(* der ausgabestring muss nochg mit 0 abgeschlossen werden *)
pt^ := 0;

(* revision history
hm		9.6.2007	rev 1.0		
	original version

hm		15.dec 2007	rev 1.1
	changed code for better performance

hm	29. mar. 2008	rev 1.2
	changed STRING to STRING(32)

hm	20. jun. 2008	rev 1.3
	performance improvement

*)

END_FUNCTION

// oscat_basic/POUs/String/DWORD_TO_STRF
FUNCTION DWORD_TO_STRF : STRING(20)
VAR_INPUT
	IN : DWORD;
	N : INT;
END_VAR


(*
version 1.0	26 jan 2007
programmer 	hugo
tested by		tobias

dword_to_strF converts a DWORD, BYTE or Word to a fixed length String.
the string will be filled with leading zeroes to achieve the fixed length, or if too long, the lowest digits will be used.
the maximum allowed length is 20 mdigits.

for example:	dword_to_strf(123,4) = '0123' 
				dword_to_strf(123,2) = '23'
*)

(* limit N to max 20 characters *)
(* convert dword to string first and cut to length N *)
DWORD_TO_STRF := FIX(DWORD_TO_STRING(in),LIMIT(0,N,20),48,1);


(* revision history
hm	26. jan.2007	rev 1.0		
	original version

hm	29. mar. 2008	rev 1.1
	changed STRING to STRING(20)
	limit the output string to max 20 digits
*)

END_FUNCTION

// oscat_basic/POUs/String/FIX
FUNCTION FIX : STRING(STRING_LENGTH)
VAR_INPUT
	str : STRING(STRING_LENGTH);
	L : INT;
	C : BYTE;
	M : INT;
END_VAR
VAR
	N : INT;
	SX: STRING(STRING_LENGTH);
END_VAR

(*
version 1.0	29. mar. 2008
programmer 	hugo
tested by	tobias

the function fix truncates a string at length L 
or if the string is shorter then L it will be filled with ending Spaces till its length = N.

*)

(* make sure L does not exceed the limits of a string *)
N := LIMIT(0,L,STRING_LENGTH) - LEN(str);
IF N <= 0 THEN
	(* truncate the string at length N *)
	IF M = 1 THEN
		FIX := RIGHT(str,L);
	ELSE
		FIX := LEFT(str,L);
	END_IF;
ELSIF M = 1 THEN
	(* connect fill characters at the beginning *)
	sx := FILL(C,N);
	FIX := CONCAT(sx,str);
ELSIF M = 2 THEN
	(* center str beween fill characters *)
	(* for an uneven number of fill characters, there is one more at the end *)
	sx := FILL(C,SHR(N+1,1));
	FIX := CONCAT(str,sx);
	SX := LEFT(sx,SHR(N,1));
	FIX := CONCAT(sx,FIX);
ELSE
	(* connect fill characters at the end *)
	SX := FILL(C,N);
	FIX := CONCAT(str,SX);
END_IF;


(* revision histroy
hm	29. mar. 2008	rev 1.0
	original release

*)

END_FUNCTION

// oscat_basic/POUs/String/DWORD_TO_STRH
FUNCTION DWORD_TO_STRH : STRING(8)
VAR_INPUT
	IN : DWORD;
END_VAR
VAR
	i : INT;
	temp : BYTE;
	pt : POINTER TO BYTE;
END_VAR

(*
version 1.3	29. mar. 2008
programmer 	hugo
tested by	tobias

DWORD_TO_STRINGH converts a DWORD to a String of Hexadecimal represented by '0' .. '9' and 'A' .. 'F'.
The lowest order Character will be on the right and the high order Character on the left.

*)

(* read output adress to pointer *)
pt := ADR(DWORD_TO_STRH) + 8;
(* wirte the closing byte for the string *)
pt^:= 0;

(* write the 8 hex characters backwards *)
FOR i := 1 TO 8 DO;
	(* decrement the pointer *)
	pt := pt - 1;
	(* read the lowest order hex value *)
	temp := DWORD_TO_BYTE(in AND 16#0000000F);
	(* convert value to hex character *)
	IF temp <= 9 THEN temp := temp + 48; ELSE temp := temp + 55; END_IF;
	(* write character to output string *)
	PT^ := temp;
	(* shift in for nect hex character *)
	in := SHR(in,4);
END_FOR;


(* code beofre rev 1.2
FOR i := 1 TO 8 DO
	X := DWORD_TO_BYTE(in AND 2#1111);
	IF X <= 9 THEN X := X + 48; ELSE X := X + 55; END_IF;
	Cx := CHR(X);
	temp := CONCAT(Cx, temp);
	in := SHR(in,4);
END_FOR;
DWORD_TO_STRH := temp;
*)


(* revision history
hm	9. jun. 2007	rev 1.0		
	original version 

hm	11. sep. 2007	rev 1.1
	changed coding for compatibility with twincat, concat cannot support a function as an argument.

hm	15. dec. 2007	rev 1.2
	changed code for better performance

hm	29. mar. 2008	rev 1.3
	changed STRING to STRING(8)

*)

END_FUNCTION

// oscat_basic/POUs/String/EXEC
FUNCTION EXEC : STRING(STRING_LENGTH)
VAR_INPUT
	str : STRING(STRING_LENGTH);
END_VAR
VAR
	pos: INT;
	R1: REAL;
	R2: REAL;
	operator: STRING(10);
END_VAR

(*
version 1.4	29. mar. 2008
programmer 	hugo
tested by		tobias

exec executes a mathematical term and returns the result as a string
the term can only be a simple term without brackets and only one operator
allowed operastors are: (+, -, *, /, ^, sqrt, sin, cos, tan).

*)

(* extract both numbers and operator *)
EXEC := UPPERCASE(TRIM(str));

pos := FINDB_NONUM(EXEC);
IF pos > 1 THEN R1 := STRING_TO_REAL(LEFT(EXEC,pos-1)); END_IF;
R2 := STRING_TO_REAL(RIGHT(EXEC,LEN(EXEC)-pos));
EXEC := LEFT(EXEC,pos);
pos := FINDB_NUM(EXEC);
operator := RIGHT(EXEC,LEN(EXEC) - pos);
IF operator = '' AND LEN(str) = 0 THEN
	EXEC := '';
	RETURN;
ELSIF operator = '' THEN
	EXEC := str;
	RETURN;
END_IF;
IF operator = '^' THEN
	EXEC := REAL_TO_STRING(EXPT(R1, R2));
ELSIF operator = 'SQRT' THEN
	EXEC := REAL_TO_STRING(SQRT(R2));
ELSIF operator = 'SIN' THEN
	EXEC := REAL_TO_STRING(SIN(r2));
ELSIF operator = 'COS' THEN
	EXEC := REAL_TO_STRING(COS(r2));
ELSIF operator = 'TAN' THEN
	EXEC := REAL_TO_STRING(TAN(R2));
ELSIF operator = '*' THEN
	EXEC := REAL_TO_STRING(R1 * R2);
ELSIF operator = '/' THEN
	IF R2 <> 0 THEN EXEC := REAL_TO_STRING(R1 / R2); ELSE EXEC := 'ERROR'; END_IF;
ELSIF operator = '+' THEN
	EXEC := REAL_TO_STRING(r1 + r2);
ELSIF operator = '-' THEN
	EXEC := REAL_TO_STRING(r1 - r2);
ELSE
	EXEC := 'ERROR';
END_IF;

IF EXEC = 'ERROR' THEN
	RETURN;
(* some systems deliver integer instead of real *)
ELSIF FIND(EXEC,'.') = 0 THEN
	EXEC := CONCAT(EXEC, '.0');
(* some systems deliver n. instead of n.0 ! *)
ELSIF RIGHT(EXEC,1) = '.' THEN
	EXEC := CONCAT(EXEC,'0');
END_IF;


(* revision history

hm 	6.feb 2007		rev 1.1
	cos has to be written in uppercase
	divide by 0 will return an error

hm	5. mar. 2008	rev 1.2
	add a 0 to the string if a '.' is at the end of the string

hm	20. mar. 2008	rev 1.3
	make sure the function always returns a real value in the form of x.y

hm	29. mar. 2008	rev 1.4
	changed STRING to STRING(STRING_LENGTH)
*)

END_FUNCTION

// oscat_basic/POUs/String/TRIM
FUNCTION TRIM : STRING(STRING_LENGTH)
VAR_INPUT
	str : STRING(STRING_LENGTH);
END_VAR
VAR
	pos: INT;
END_VAR

(*
version 1.2	29. mar. 2008
programmer 	hugo
tested by	tobias

the function deletes all blanks within a string.

*)

TRIM := str;
REPEAT
	pos := FIND(trim,' ');
	IF pos > 0 THEN TRIM := REPLACE(TRIM,'',1,pos); END_IF;
UNTIL pos = 0	END_REPEAT;


(* revision histroy
hm	6.10.2006		rev 1.0
	original release

hm	20. mar. 2008	rev 1.1
	avoid to call replace with pos = 0 because some systems will produce an error

hm	29. mar. 2008	rev 1.2
	changed STRING to STRING(STRING_LENGTH)
*)

END_FUNCTION

// oscat_basic/POUs/String/FINDB_NONUM
FUNCTION FINDB_NONUM : INT
VAR_INPUT
	str : STRING(STRING_LENGTH);
END_VAR
VAR
	pos: INT;
	pt : POINTER TO BYTE;
END_VAR

(*
version 1.3	21. oct. 2008
programmer 	hugo
tested by	oscat

findB_noNum searches str backwards and returns the last position which is not a number.
a number is characterized by a letter "0..9" or "."

*)

pt := ADR(str) + LEN(str) - 1;
FOR pos := LEN(str) TO 1 BY -1 DO;
	IF (PT^ < 48 AND PT^ <> 46) OR PT^ > 57 THEN
		FINDB_NONUM := pos;
		RETURN;
	END_IF;
	PT := PT - 1;
END_FOR;
FINDB_NONUM := 0;


(* revision history
hm	6. oct 2006		rev 1.0
	original version

hm	29. feb 2008	rev 1.1
	improved performance

hm	29. mar. 2008	rev 1.2
	changed STRING to STRING(STRING_LENGTH)

hm	21. oct. 2008	rev 1.3
	optimized code
*)

END_FUNCTION

// oscat_basic/POUs/String/FINDB_NUM
FUNCTION FINDB_NUM : INT
VAR_INPUT
	str : STRING(STRING_LENGTH);
END_VAR
VAR
	pos: INT;
	pt : POINTER TO BYTE;
END_VAR

(*
version 1.2	29. mar. 2008
programmer 	hugo
tested by	tobias

findB_Num searches str backward and returns the last position of a number
a number is characterized by a letter "0..9" or "."

*)

pt := ADR(str) + LEN(str) - 1;
FOR pos := LEN(str) TO 1 BY -1 DO;
	IF (PT^ > 47 AND PT^ < 58) OR PT^ = 46 THEN
		FINDB_NUM := pos;
		RETURN;
	END_IF;
	PT := PT - 1;
END_FOR;
FINDB_NUM := 0;

(* revision history
hm	6. oct 2006		rev 1.0
	original version

hm	29. feb 2008	rev 1.1
	improved performance

hm	29. mar. 2008	rev 1.2
	changed STRING to STRING(STRING_LENGTH)
*)

END_FUNCTION

// oscat_basic/POUs/String/FIND_CHAR
FUNCTION FIND_CHAR : INT
VAR_INPUT
	str : STRING(STRING_LENGTH);
	pos : INT;
END_VAR
VAR
	i: INT;
	pt : POINTER TO ARRAY[1..255] OF BYTE;
	stop: INT;
	X: BYTE;
END_VAR

(*
version 1.3	21. oct. 2008
programmer 	hugo
tested by	tobias

find_char searches str and returns the starting position of the first character that is not a control character.
control characters are the ascii character 00 .. 31 and 127

*)

pt := ADR(str);
stop := LEN(str);
FOR i := MAX(pos,1) TO stop DO;
	X := pt^[i];
	IF X > 31 AND ((setup.EXTENDED_ASCII AND X <> 127) OR (NOT setup.EXTENDED_ASCII AND X < 127)) THEN
		FIND_CHAR := i;
		RETURN;
	END_IF;
END_FOR;
FIND_CHAR := 0;


(* revision history
hm	29. feb 2008	rev 1.0
	original version

hm	26. mar. 2008	rev 1.1
	char will now accept extended ascii

hm	29. mar. 2008	rev 1.2
	changed STRING to STRING(STRING_LENGTH)

hm	21. oct. 2008	rev 1.3
	changes setup constants
	optimized code
*)

END_FUNCTION

// oscat_basic/POUs/String/FIND_CTRL
FUNCTION FIND_CTRL : INT
VAR_INPUT
	str : STRING(STRING_LENGTH);
	pos : INT;
END_VAR
VAR
	i: INT;
	pt : POINTER TO ARRAY[1..255] OF BYTE;
	stop: INT;
	x: BYTE;
END_VAR

(*
version 1.2	29. mar. 2008
programmer 	hugo
tested by		tobias

find_ctrl searches str and returns the starting position of a control character
control characters are the ascii character 00 .. 31 and 127.

*)

pt := ADR(str);
stop := LEN(str);
FOR i := MAX(pos,1) TO stop DO;
	x := PT^[I];
	IF x < 32 OR X = 127 THEN
		FIND_CTRL := i;
		RETURN;
	END_IF;
END_FOR;
FIND_CTRL := 0;


(* revision history
hm	29. feb 2008	rev 1.0
	original version

hm	26. mar. 2008	rev 1.1
	character 127 is now recognized as control

hm	29. mar. 2008	rev 1.2
	changed STRING to STRING(STRING_LENGTH)
*)

END_FUNCTION

// oscat_basic/POUs/String/FIND_NONUM
FUNCTION FIND_NONUM : INT
VAR_INPUT
	str : STRING(STRING_LENGTH);
	pos : INT;
END_VAR
VAR
	i: INT;
	pt : POINTER TO ARRAY[1..255] OF BYTE;
	end: INT;
	X: BYTE;
END_VAR

(*
version 1.3	21. oct. 2008
programmer 	hugo
tested by	tobias

find_noNum searches str and returns the first position which is not a number.
a number is characterized by a letter "0..9" or "."

*)

pt := ADR(str);
end := LEN(str);
FOR i := MAX(pos,1) TO end DO;
	X := pt^[i];
	IF (X < 48 AND X <> 46) OR X > 57 THEN
		FIND_NONUM := i;
		RETURN;
	END_IF;
END_FOR;
FIND_NONUM := 0;


(* revision history
hm	6. oct. 2006	rev 1.0
	original version

hm	29. feb 2008	rev 1.1
	added input pos to start search at position

hm	29. mar. 2008	rev 1.2
	changed STRING to STRING(STRING_LENGTH)

hm	21. oct. 2008	rev 1.3
	optimized code

*)

END_FUNCTION

// oscat_basic/POUs/String/FIND_NUM
FUNCTION FIND_NUM : INT
VAR_INPUT
	str : STRING(STRING_LENGTH);
	pos : INT;
END_VAR
VAR
	i : INT;
	pt : POINTER TO ARRAY[1..255] OF BYTE;
	stop : INT;
	X: BYTE;
END_VAR

(*
version 1.2	29. mar. 2008
programmer 	hugo
tested by		tobias

find_Num searches str and returns the starting position of a number
a number is characterized by a letter "0..9" or "."

*)

pt := ADR(str);
stop := LEN(str);
FOR i := MAX(pos,1) TO stop DO;
	X := pt^[i];
	IF (X > 47 AND X < 58) OR X = 46 THEN
		FIND_NUM := i;
		RETURN;
	END_IF;
END_FOR;
FIND_NUM := 0;


(* revision history
hm	6. oct. 2006	rev 1.0
	original version

hm	29. feb 2008	rev 1.1
	added input pos to start search at position

hm	29. mar. 2008	rev 1.2
	changed STRING to STRING(STRING_LENGTH)

*)

END_FUNCTION

// oscat_basic/POUs/String/FINDB
FUNCTION FINDB : INT
VAR_INPUT
	str1 : STRING(STRING_LENGTH);
	str2 : STRING(STRING_LENGTH);
END_VAR
VAR
	pos: INT;
	length: INT;
END_VAR

(*
version 1.3	29. mar. 2008
programmer 	hugo
tested by		tobias

the function find searches an str1 for the presence of str2 and returns the first position of str1 of the last presence in instring.
the function is similar to find except it searches from the right to left.
 a 0 is returned if the string is not found.

*)

length := LEN(str2);
FOR pos := LEN(str1) - length + 1 TO 1 BY -1 DO
	IF MID(str1,length,pos) = str2 THEN
		FindB := pos;
		RETURN;
	END_IF;
END_FOR;
FindB := 0;

(* revision history
hm	6. oct 2006		rev 1.0
	original version

hm	15 dec 2007		rev 1.1
	changed code for better performance

hm	29. feb 2008	rev 1.2
	added findb := 0 for compatibility reasons

hm	29. mar. 2008	rev 1.3
	changed STRING to STRING(STRING_LENGTH)
*)

END_FUNCTION

// oscat_basic/POUs/String/FINDP
FUNCTION FINDP : INT
VAR_INPUT
	str : STRING(STRING_LENGTH);
	src : STRING(STRING_LENGTH);
	pos: INT;
END_VAR
VAR
	i: INT;
	ls: INT;
	lx: INT;
	stp: INT;
END_VAR

(*
version 1.2	29. mar. 2008
programmer 	hugo
tested by	tobias

the function findP searches a string str for the occurence of src beginning at the position pos.

*)

ls := LEN(str);
lx := LEN(src);
IF ls < lx OR lx = 0 THEN RETURN; END_IF;
stp := ls - lx + 1;
FOR i := MAX(pos,1) TO stp DO
	IF MID(str,lx,i) = src THEN
		FINDP := i;
		RETURN;
	END_IF;
END_FOR;
FINDP := 0;

(* revision histroy
hm	4. feb. 2008	rev 1.0
	original release

hm	29. feb 2008	rev 1.1
	ADDED MAX(pos,1) in loop initialization

hm	29. mar. 2008	rev 1.2
	changed STRING to STRING(STRING_LENGTH)
*)

END_FUNCTION

// oscat_basic/POUs/String/FLOAT_TO_REAL
FUNCTION FLOAT_TO_REAL : REAL
VAR_INPUT
	FLT : STRING(20);
END_VAR
VAR
	pt : POINTER TO ARRAY[1..20] OF BYTE;
	i: INT;
	X: BYTE;
	sign: INT := 1;
	stop: INT;
	tmp: DINT;
	d : INT;
END_VAR

(*
version 1.3	23. oct. 2008
programmer 	hugo
tested by	oscat

FLOAT_TO_REAL converts a string to a REAL.
the function ignores all wrong characters.
the comma can be , or .
the exponent has to start with capital E or lowercase e .


*)

pt := ADR(FLT);
stop := LEN(FLT);

(* we first check for sign and exit if first number or dot is reached *)
FOR i := 1 TO stop DO
	X := pt^[i];
	IF X > 47 AND X < 58 OR X = 46 THEN
		EXIT;
	ELSIF X = 45 THEN
		(* code 45 is sign *)
		sign := -1;
	END_IF;
END_FOR;

(* now we scan numbers till end or dot or E is reached *)
FOR i := i TO stop DO
	X := pt^[i];
	IF X = 44 OR X = 46 OR X = 69 OR X = 101 THEN
		EXIT;
	(* calculate the value of the digit *)
	ELSIF X > 47 AND x < 58 THEN
		tmp := tmp * 10 + X - 48;
	END_IF;
END_FOR;

(* process the portion after the comma if comma or dot is reached exit if exponent starts *)
IF x = 44 OR X = 46 THEN
	FOR i := i + 1 TO stop DO
		X := pt^[i];
		IF X = 69 OR X = 101 THEN
			EXIT;
		ELSIF x > 47 AND x < 58 THEN
			tmp := tmp * 10 + X - 48;
			d := d - 1;
		END_IF;
	END_FOR;
END_IF;

(* process exponent if present *)
IF X = 69 OR X = 101 THEN
	d := d + DEC_TO_INT(RIGHT(FLT, stop - i));
END_IF;

FLOAT_TO_REAL :=  EXPN(10, d) * DINT_TO_REAL(TMP * SIGN);




(* revision histroy
hm	22. jun. 2008	rev 1.0
	original release

hm	2. oct. 2008	rev 1.1
	fixed an error, characters 8 and 9 would not be converted

hm	22. oct. 2008	rev 1.2
	last fix was not done correctly

hm	23. oct. 2008	rev 1.3
	optimzed code
*)

END_FUNCTION

// oscat_basic/POUs/String/FSTRING_TO_BYTE
FUNCTION FSTRING_TO_BYTE : BYTE
VAR_INPUT
	IN : STRING(12);
END_VAR


(*
version 1.1	20. sep. 2008
programmer 	hugo
tested by		oscat

FSTRING_TO_BYTE converts a formatted string into a byte.
the string can be of the form 2#01010, 8#7234, 16#2AD3 and 1234

*)

IF LEFT(IN, 2) = '2#' THEN
	(* we need to convert binary *)
	FSTRING_TO_BYTE := BIN_TO_BYTE(RIGHT(in, LEN(in) - 2));
ELSIF LEFT(in, 2) = '8#' THEN
	(* weneed to convert octals *)
	FSTRING_TO_BYTE := OCT_TO_BYTE(RIGHT(in, LEN(in) - 2));
ELSIF LEFT(in, 3) = '16#' THEN
	(* we need to convert hexadecimal *)
	FSTRING_TO_BYTE := HEX_TO_BYTE(RIGHT(in, LEN(in) - 3));
ELSE
	(* we assume decimal representation *)
	FSTRING_TO_BYTE := DEC_TO_BYTE(CLEAN(in,'0123456789'));
END_IF;


(* revision histroy
hm	18. jun. 2008	rev 1.0
	original release

hm	20. sep. 2008	rev 1.1
	changed length of input string from 20 to 12
*)

END_FUNCTION

// oscat_basic/POUs/String/OCT_TO_BYTE
FUNCTION OCT_TO_BYTE : BYTE
VAR_INPUT
	OCT : STRING(10);
END_VAR
VAR
	pt : POINTER TO BYTE;
	i: INT;
	X: BYTE;
	stop: INT;
END_VAR

(*
version 1.1	20. sep. 2008
programmer 	hugo
tested by		oscat

OCT_TO_BYTE converts a octagonal string into a byte.

*)

pt := ADR(oct);
stop := LEN(oct);
FOR I := 1 TO stop DO
	(* read the first character and subtract 48 to get value in decimal 0 = 48 *)
	x := pt^;
	(* calculate the value of the digit *)
	IF X > 47 AND x < 56 THEN
		OCT_TO_BYTE := SHL(OCT_TO_BYTE,3) + X - 48;
	END_IF;
	pt := pt + 1;
END_FOR;



(* revision histroy
hm	18. jun. 2008	rev 1.0
	original release

hm	20. sep. 2008	rev 1.1
	changed length of input string from 20 to 10

*)

END_FUNCTION

// oscat_basic/POUs/String/HEX_TO_BYTE
FUNCTION HEX_TO_BYTE : BYTE
VAR_INPUT
	HEX : STRING(5);
END_VAR
VAR
	pt : POINTER TO BYTE;
	i: INT;
	X: BYTE;
	stop: INT;
END_VAR

(*
version 1.1	20. sep. 2008
programmer 	hugo
tested by		oscat

HEX_TO_BYTE converts a Hexadecimal string into a byte.

*)

pt := ADR(hex);
stop := LEN(hex);
FOR I := 1 TO stop DO
	(* read the first character and subtract 48 to get value in decimal 0 = 48 *)
	x := pt^;
	(* calculate the value of the digit *)
	IF X > 47 AND x < 58 THEN
		HEX_TO_BYTE := SHL(HEX_TO_BYTE,4) + X - 48;
	ELSIF X > 64 AND X < 71 THEN
		HEX_TO_BYTE := SHL(HEX_TO_BYTE,4) + X - 55;
	ELSIF X > 96 AND X < 103 THEN
		HEX_TO_BYTE := SHL(HEX_TO_BYTE,4) + X - 87;
	END_IF;
	pt := pt + 1;
END_FOR;




(* revision histroy
hm	18. jun. 2008	rev 1.0
	original release

hm	20. sep.2008	rev 1.1
	changed length of input string from 20 to 5

*)

END_FUNCTION

// oscat_basic/POUs/String/FSTRING_TO_DT
FUNCTION FSTRING_TO_DT : DT
VAR_INPUT
	SDT : STRING(60);
	FMT : STRING(60);
END_VAR
VAR CONSTANT
	ignore: STRING(1) := '*';  (* ignore character is * *)
	fchar : STRING(1) := '#';  (* format character is # *)
END_VAR
VAR
	c: STRING(1);
	tmp: STRING(20);
	end: INT;
	dy : INT := 1970;
	dm : INT := 1;
	dd : INT := 1;
	th : INT;
	tm : INT;
	ts : INT;
END_VAR


(*
version 1.0	24. sep. 2008
programmer 	hugo
tested by	oscat

FSTRING_TO_DT converts Formatted String into a DT value.

*)

(* scan input string *)
WHILE fmt <> '' DO
	c := LEFT(fmt,1);
	IF c = ignore THEN
		(* skip ignore characters *)
		fmt := DELETE(fmt,1,1);
		sdt := DELETE(sdt,1,1);
	ELSIF C = fchar THEN
		(* format chracter found skip format char and read identifier *)
		(* store format identifier in c and skip to next char in fmt *)
		c := MID(fmt,1,2);
		fmt := DELETE(fmt,2,1);
		(* extract the substring until the end of sdt or to next char of fmt *)
		IF fmt = '' THEN
			tmp := sdt;
		ELSE
			(* serach for end of substring *)
			end := FIND(sdt, LEFT(fmt,1))-1;
			tmp := LEFT(sdt, end);
			sdt := DELETE(sdt, end,1);
		END_IF;
		(* extract information from substring *)
		IF c = 'Y' THEN
			dy := STRING_TO_INT(tmp);
			IF dy < 100 THEN dy := dy + 2000; END_IF;
		ELSIF c = 'M' THEN
			dm := STRING_TO_INT(tmp);
		ELSIF c = 'N' THEN
			dm := FSTRING_TO_MONTH(tmp,0);
		ELSIF c = 'D' THEN
			dd := STRING_TO_INT(tmp);
		ELSIF c = 'h' THEN
			th := STRING_TO_INT(tmp);
		ELSIF c = 'm' THEN
			tm := STRING_TO_INT(tmp);
		ELSIF c = 's' THEN
			ts := STRING_TO_INT(tmp);
		END_IF;
	ELSIF c = LEFT(sdt,1) THEN
		(* skip matching characters *)
		fmt := DELETE(fmt,1,1);
		sdt := DELETE(sdt,1,1);
	ELSE
		RETURN;
	END_IF;
END_WHILE;

FSTRING_TO_DT := SET_DT(dy,dm,dd,th,tm,ts);


(* revision histroy
hm	24. sep. 2008	rev 1.0
	original release


*)

END_FUNCTION

// oscat_basic/POUs/String/FSTRING_TO_MONTH
FUNCTION FSTRING_TO_MONTH : INT
VAR_INPUT
	MTH : STRING(20);
	LANG : INT;
END_VAR
VAR
	lx: INT;
END_VAR


(*
version 1.2	25. oct 2008
programmer 	hugo
tested by	oscat

FSTRING_TO_MONTH converts a string into a month, the string can be a name for the month or a number.
the function is language sensitve when LANG > 1 and checks for all languages when LANG = 0

*)

IF LANG = 0 THEN lx := LANGUAGE.DEFAULT; ELSE lx := MIN(LANG, LANGUAGE.LMAX); END_IF;
MTH := TRIM(mth);
MTH := CAPITALIZE(LOWERCASE(MTH));

FOR FSTRING_TO_MONTH := 1 TO 12 DO
	IF MTH = language.MONTHS[lx, FSTRING_TO_MONTH] THEN RETURN; END_IF;
	IF MTH = language.MONTHS3[lx, FSTRING_TO_MONTH] THEN RETURN; END_IF;
END_FOR;

(* since no name matched try to decode as integer *)
FSTRING_TO_MONTH := STRING_TO_INT(MTH);




(* revision histroy
hm	25. sep. 2008	rev 1.0
	original release

hm	19. oct. 2008	rev 1.1
	changed language setup constants

hm	25. oct. 2008	rev 1.2
	optimized code
*)

END_FUNCTION

// oscat_basic/POUs/Time&Date/SET_DT
FUNCTION SET_DT : DT
VAR_INPUT
	year : INT;
	month : INT;
	day : INT;
	hour : INT;
	minute : INT;
	second : INT;
END_VAR


(*
version 1.5	16 mar 2008
programmer 	hugo
tested by	tobias


creates a date output from year, month and day of month
year must be in the form of 4 digits ie 2006 or 1977.
*)

SET_DT := DWORD_TO_DT(DATE_TO_DWORD(SET_DATE(YEAR, MONTH, day)) + INT_TO_DWORD(SECOND) + INT_TO_DWORD(MINUTE) * 60 + INT_TO_DWORD(HOUR) * 3600);


(* revision history
hm	4. aug. 2006		rev 1.0
	original version

hm		19 sep. 2007	rev 1.1
	use function leap_year to calculate leap year, more exceptions are handled

hm		1. okt 2007		rev 1.2
	added step7 compatibility
	call function set_date

hm		8. oct 2007		rev 1.3
	deleted unused variables count and leap

hm		1. 11 2007		rev 1.4
	converted hour type integer to dword in calculation to avoid overrun on möller ecp4

hm		16. mar 2008	rev 1.5
	added type conversions to avoid warnings under codesys 3.0
*)

END_FUNCTION

// oscat_basic/POUs/String/FSTRING_TO_DWORD
FUNCTION FSTRING_TO_DWORD : DWORD
VAR_INPUT
	IN : STRING(40);
END_VAR


(*
version 1.1	20. sep. 2008
programmer 	hugo
tested by		oscat

FSTRING_TO_BYTE converts a formatted string into a byte.
the string can be of the form 2#01010, 8#7234, 16#2AD3 and 1234

*)

IF LEFT(IN, 2) = '2#' THEN
	(* we need to convert binary *)
	FSTRING_TO_DWORD := BIN_TO_DWORD(RIGHT(in, LEN(in) - 2));
ELSIF LEFT(in, 2) = '8#' THEN
	(* weneed to convert octals *)
	FSTRING_TO_DWORD := OCT_TO_DWORD(RIGHT(in, LEN(in) - 2));
ELSIF LEFT(in, 3) = '16#' THEN
	(* we need to convert hexadecimal *)
	FSTRING_TO_DWORD := HEX_TO_DWORD(RIGHT(in, LEN(in) - 3));
ELSE
	(* we assume decimal representation *)
	FSTRING_TO_DWORD := DEC_TO_DWORD(CLEAN(in,'0123456789'));
END_IF;


(* revision histroy
hm	18. jun. 2008	rev 1.0
	original release

hm	20. sep. 2008	rev 1.1
	changed length of input dtring from 20 to 40


*)

END_FUNCTION

// oscat_basic/POUs/String/OCT_TO_DWORD
FUNCTION OCT_TO_DWORD : DWORD
VAR_INPUT
	OCT : STRING(20);
END_VAR
VAR
	pt : POINTER TO BYTE;
	i: INT;
	X: BYTE;
	stop: INT;
END_VAR

(*
version 1.0	18. jun 2008
programmer 	hugo
tested by	oscat

OCT_TO_DWORD converts a octagonal string into a dword.

*)

pt := ADR(oct);
stop := LEN(oct);
FOR I := 1 TO stop DO
	(* read the first character and subtract 48 to get value in decimal 0 = 48 *)
	x := pt^;
	(* calculate the value of the digit *)
	IF X > 47 AND x < 56 THEN
		OCT_TO_DWORD := SHL(OCT_TO_DWORD,3) + X - 48;
	END_IF;
	pt := pt + 1;
END_FOR;




(* revision histroy
hm	18. jun. 2008	rev 1.0
	original release


*)

END_FUNCTION

// oscat_basic/POUs/String/HEX_TO_DWORD
FUNCTION HEX_TO_DWORD : DWORD
VAR_INPUT
	Hex : STRING(20);
END_VAR
VAR
	pt : POINTER TO BYTE;
	i: INT;
	X: BYTE;
	stop: INT;
END_VAR

(*
version 1.4	18. jun. 2008
programmer 	hugo
tested by	tobias

HEX_TO_DWORD converts a Hexadecimal string into a DWORD.

*)

pt := ADR(hex);
stop := LEN(hex);
FOR I := 1 TO stop DO
	(* read the first character and subtract 48 to get value in decimal 0 = 48 *)
	x := pt^;
	(* calculate the value of the digit *)
	IF X > 47 AND x < 58 THEN
		HEX_TO_DWORD := SHL(HEX_TO_DWORD,4) + X - 48;
	ELSIF X > 64 AND X < 71 THEN
		HEX_TO_DWORD := SHL(HEX_TO_DWORD,4) + X - 55;
	ELSIF X > 96 AND X < 103 THEN
		HEX_TO_DWORD := SHL(HEX_TO_DWORD,4) + X - 87;
	END_IF;
	pt := pt + 1;
END_FOR;



(* revision histroy
hm	2.10.2007		rev 1.0
	original release

hm	19.11.2007		rev 1.1
	changed type of function from int to dword

hm 	4. mar 2008		rev 1.2
	added support for a..f and return 0 for invalid string

hm	29. mar. 2008	rev 1.3
	changed STRING to STRING(8)

hm	18. jun. 2008	rev 1.4
	changed input hex to STRING(20)
	function now ignores wrong characters
*)

END_FUNCTION

// oscat_basic/POUs/String/FSTRING_TO_WEEK
FUNCTION FSTRING_TO_WEEK : BYTE
VAR_INPUT
	WEEK : STRING(60);
	LANG : INT;
END_VAR
VAR
	pos: INT;
END_VAR


(*
version 1.1	25. oct. 2008
programmer 	hugo
tested by	oscat

FSTRING_TO_WEEK converts a list of weekdays into a byte where each bit represents a day of the week.
bit 6 = mo, 0 = su;

*)

pos := FIND(WEEK, ',');
WHILE pos > 0 DO
	FSTRING_TO_WEEK := FSTRING_TO_WEEK OR SHR(BYTE#128, FSTRING_TO_WEEKDAY(MID(WEEK, pos - 1, 1), LANG));
	WEEK := RIGHT(WEEK, LEN(Week) - pos);
	pos := FIND(WEEK, ',');
END_WHILE;
FSTRING_TO_WEEK := (FSTRING_TO_WEEK OR SHR(BYTE#128, FSTRING_TO_WEEKDAY(WEEK, LANG))) AND BYTE#127;


(* revision histroy
hm	18. jun. 2008	rev 1.0
	original release

hm	25. oct. 2008	rev 1.1
	using language defauls and input lang
*)

END_FUNCTION

// oscat_basic/POUs/String/FSTRING_TO_WEEKDAY
FUNCTION FSTRING_TO_WEEKDAY : INT
VAR_INPUT
	WDAY : STRING(20);
	LANG : INT;
END_VAR
VAR
	tmp: STRING(2);
	i: INT;
	ly: INT;
END_VAR


(*
version 1.2	25. oct. 2008
programmer 	hugo
tested by	oscat

FSTRING_TO_WEEKDAY converts a weekday string into an integer 1..7.

*)

IF LANG = 0 THEN ly := LANGUAGE.DEFAULT; ELSE ly := MIN(LANG, LANGUAGE.LMAX); END_IF;
(* tmp needs to be calculated first otherwise find can return wrong values *)
tmp := TRIM(wday);
tmp := CAPITALIZE(LOWERCASE(tmp));
FOR i := 1 TO 7 DO
	IF language.WEEKDAYS2[ly, i] = tmp THEN
		FSTRING_TO_WEEKDAY := i;
		RETURN;
	END_IF;
END_FOR;
FSTRING_TO_WEEKDAY := STRING_TO_INT(WDAY);




(* revision histroy
hm	18. jun. 2008	rev 1.0
	original release

hm	18. jul. 2008	rev 1.1
	changed nested call of left(trim()) for compatibility reasons

hm	25. oct. 2008	rev 1.2
	using language constants
*)

END_FUNCTION

// oscat_basic/POUs/String/IS_ALNUM
FUNCTION IS_ALNUM : BOOL
VAR_INPUT
	str : STRING(STRING_LENGTH);
END_VAR
VAR
	L: INT;
	pt : POINTER TO BYTE;
	pos: INT;
END_VAR

(*
version 1.1	29. mar. 2008
programmer 		kurt
tested by		hugo

ISC_ALNUM testet ob in einem string nur Zahlen 0..9 vorkommen.

*)

PT := ADR(str);
L := LEN(str);
FOR pos := 1 TO L DO
	IF NOT (ISC_ALPHA(pt^) OR ISC_NUM(pt^)) THEN
		IS_ALNUM := FALSE;
		RETURN;
	END_IF;
    	PT := PT + 1;
END_FOR;
IS_ALNUM := L > 0;


(* revision history
hm	29. feb 2008	rev 1.0
	original version

hm	29. mar. 2008	rev 1.1
	changed STRING to STRING(STRING_LENGTH)
*)

END_FUNCTION

// oscat_basic/POUs/String/ISC_ALPHA
FUNCTION ISC_ALPHA : BOOL
VAR_INPUT
	IN : BYTE;
END_VAR


(*
version 1.1	19. oct. 2008
programmer 	oscat
tested by	oscat

ISC_ALPHA checks if a character is a..z or A..Z.

*)

IF setup.EXTENDED_ASCII THEN
	ISC_ALPHA := (in > 64 AND in < 91) OR (in > 191  AND in <> 215 AND in <> 247) OR (in > 96 AND in < 123);
ELSE
	ISC_ALPHA := (IN > 64 AND IN < 91) OR (in > 96 AND in < 123);
END_IF;

(* revision history
hm	6. mar. 2008	rev 1.0
	original version

hm	19. oct. 2008	rev 1.1
	changes setup constants
*)

END_FUNCTION

// oscat_basic/POUs/String/ISC_NUM
FUNCTION ISC_NUM : BOOL
VAR_INPUT
	IN : BYTE;
END_VAR


(*
version 1.0	6. mar 2008
programmer 	oscat
tested by		hugo

ISC_NUM checks if a character is 0..9.

*)

ISC_NUM := IN > 47 AND IN < 58;

(* revision history
hm		6. mar. 2008	rev 1.0
	original version

*)

END_FUNCTION

// oscat_basic/POUs/String/IS_ALPHA
FUNCTION IS_ALPHA : BOOL
VAR_INPUT
	str : STRING(STRING_LENGTH);
END_VAR
VAR
	L: INT;
	pt : POINTER TO BYTE;
	pos: INT;
END_VAR

(*
version 1.1	29. mar. 2008
programmer 		kurt
tested by		hugo

IS_ALPHA testet ob in einem string nur Zeichen a-z oder A - Z vorkommen.

*)

PT := ADR(str);
L := LEN(str);
FOR pos := 1 TO L DO
	IF NOT ISC_ALPHA(pt^) THEN
		IS_ALPHA := FALSE;
		RETURN;
	END_IF;
    	PT := PT + 1;
END_FOR;
IS_ALPHA := L > 0;


(* revision history
hm	29. feb 2008	rev 1.0
	original version

hm	29. mar. 2008	rev 1.1
	changed STRING to STRING(STRING_LENGTH)
*)

END_FUNCTION

// oscat_basic/POUs/String/IS_CC
FUNCTION IS_CC : BOOL
VAR_INPUT
	str : STRING(STRING_LENGTH);
	cmp : STRING(STRING_LENGTH);
END_VAR
VAR
	L: INT;
	pos: INT;
END_VAR

(*
version 1.1	29. mar. 2008
programmer 	Tobias
tested by	hugo

ISC_CC testet ob ein string nur aus Zeichen des Strings CMP besteht.

*)

L := LEN(str);
FOR pos := 1 TO L DO
	IF FIND(CMP,MID(str,1,pos)) = 0 THEN RETURN; END_IF;
END_FOR;
IS_CC := L > 0;



(* revision history
hm	19. mar 2008	rev 1.0
	original version

hm	29. mar. 2008	rev 1.1
	changed STRING to STRING(STRING_LENGTH)
*)

END_FUNCTION

// oscat_basic/POUs/String/IS_CTRL
FUNCTION IS_CTRL : BOOL
VAR_INPUT
	STR : STRING(STRING_LENGTH);
END_VAR
VAR
	L: INT;
	pt : POINTER TO BYTE;
	pos: INT;
END_VAR

(*
version 1.1	29. mar 2008
programmer 		kurt
tested by		hugo

IS_CTRL testet ob in einem string nur Steuerzeichen (Char < 32) vorkommen.

*)

PT := ADR(str);
L := LEN(str);
FOR pos := 1 TO L DO
	IF NOT (ISC_CTRL(pt^)) THEN
		IS_CTRL := FALSE;
		RETURN;
	END_IF;
    	PT := PT + 1;
END_FOR;
IS_CTRL := L > 0;


(* revision history
hm	29. feb. 2008	rev 1.0
	original version

hm	29. mar. 2008	rev 1.1
	changed STRING to STRING(STRING_LENGTH)
*)

END_FUNCTION

// oscat_basic/POUs/String/ISC_CTRL
FUNCTION ISC_CTRL : BOOL
VAR_INPUT
	IN : BYTE;
END_VAR


(*
version 1.0	6. mar 2008
programmer 	oscat
tested by		hugo

ISC_ALPHA checks if a character is a control character.

*)

ISC_CTRL := IN < 32 OR IN = 127;

(* revision history
hm		6. mar. 2008	rev 1.0
	original version

*)

END_FUNCTION

// oscat_basic/POUs/String/IS_HEX
FUNCTION IS_HEX : BOOL
VAR_INPUT
	str : STRING(STRING_LENGTH);
END_VAR
VAR
	L: INT;
	pt : POINTER TO BYTE;
	pos: INT;
END_VAR

(*
version 1.1	29. mar. 2008
programmer 		kurt
tested by		hugo

IS_HEX testet ob in einem string nur Zahlen 0..9 oder A..F oder a..f  vorkommen.

*)

PT := ADR(str);
L := LEN(str);
FOR pos := 1 TO L DO
	IF NOT (ISC_HEX(pt^)) THEN
		IS_HEX := FALSE;
		RETURN;
	END_IF;
    	PT := PT + 1;
END_FOR;
IS_HEX := L > 0;


(* revision history
hm	29. feb 2008	rev 1.0
	original version

hm	29. mar. 2008	rev 1.1
	changed STRING to STRING(STRING_LENGTH)
*)

END_FUNCTION

// oscat_basic/POUs/String/ISC_HEX
FUNCTION ISC_HEX : BOOL
VAR_INPUT
	IN : BYTE;
END_VAR


(*
version 1.0	6. mar 2008
programmer 	oscat
tested by		hugo

ISC_HEX checks if a character is 0..9, A..F, a..f.

*)

ISC_HEX := (IN > 47 AND IN < 58) OR (IN > 64 AND IN < 71) OR (IN > 96 AND IN < 103);

(* revision history
hm		6. mar. 2008	rev 1.0
	original version

*)

END_FUNCTION

// oscat_basic/POUs/String/IS_LOWER
FUNCTION IS_LOWER : BOOL
VAR_INPUT
	str : STRING(STRING_LENGTH);
END_VAR
VAR
	l: INT;
	pt : POINTER TO BYTE;
	pos: INT;
END_VAR

(*
version 1.1	29. mar. 2008
programmer 		kurt
tested by		hugo

IS_LOWER testet ob in einem string nur kleinbuchstaben vorkommen.

*)

PT := ADR(str);
L := LEN(str);
FOR pos := 1 TO L DO
	IF NOT (ISC_LOWER(pt^)) THEN
		IS_LOWER := FALSE;
		RETURN;
	END_IF;
    	PT := PT + 1;
END_FOR;
IS_LOWER := L > 0;


(* revision history
hm	29. feb 2008	rev 1.0
	original version

hm	29. mar. 2008	rev 1.1
	changed STRING to STRING(STRING_LENGTH)
*)

END_FUNCTION

// oscat_basic/POUs/String/ISC_LOWER
FUNCTION ISC_LOWER : BOOL
VAR_INPUT
	IN : BYTE;
END_VAR


(*
version 1.1	19. oct. 2008
programmer 	hugo
tested by	oscat

isc_lower checks if a character is lowercase.

*)

IF setup.EXTENDED_ASCII THEN
	ISC_LOWER := ((in > 96) AND (in < 123)) OR ((in > 222) AND (in <> 247));
ELSE
	ISC_LOWER := ((in > 96) AND (in < 123));
END_IF;

(* revision history
hm	6. mar. 2008	rev 1.0
	original version

hm	19. oct. 2008	rev 1.1
	changes setup constants
*)

END_FUNCTION

// oscat_basic/POUs/String/IS_NCC
FUNCTION IS_NCC : BOOL
VAR_INPUT
	str : STRING(STRING_LENGTH);
	cmp : STRING(STRING_LENGTH);
END_VAR
VAR
	L: INT;
	pos: INT;
END_VAR

(*
version 1.1	29. mar. 2008
programmer 	Tobias
tested by		hugo

IS_NCC testet ob in einem string keine Zeichen des Strings CMP enthalten sind.

*)

L := LEN(str);
FOR pos := 1 TO L DO
	IF FIND(CMP,MID(str,1,pos)) > 0 THEN RETURN; END_IF;
END_FOR;
IS_NCC := TRUE;



(* revision history
hm	19. mar 2008	rev 1.0
	original version

hm	29. mar. 2008	rev 1.1
	changed STRING to STRING(STRING_LENGTH)
*)

END_FUNCTION

// oscat_basic/POUs/String/IS_NUM
FUNCTION IS_NUM : BOOL
VAR_INPUT
	str : STRING(STRING_LENGTH);
END_VAR
VAR
	L : INT;
	pt : POINTER TO BYTE;
	pos: INT;
END_VAR

(*
version 1.1	29. mar. 2008
programmer 		kurt
tested by		hugo

IS_NUM testet ob in einem string nur Zahlen 0..9 vorkommen.

*)

PT := ADR(str);
L := LEN(str);
FOR pos := 1 TO L DO
	IF NOT (ISC_NUM(pt^)) THEN
		IS_NUM := FALSE;
		RETURN;
	END_IF;
    	PT := PT + 1;
END_FOR;
IS_NUM := L > 0;


(* revision history
hm	29. feb 2008	rev 1.0
	original version

hm	29. mar. 2008	rev 1.1
	changed STRING to STRING(STRING_LENGTH)
*)

END_FUNCTION

// oscat_basic/POUs/String/IS_UPPER
FUNCTION IS_UPPER : BOOL
VAR_INPUT
	str : STRING(STRING_LENGTH);
END_VAR
VAR
	L: INT;
	pt : POINTER TO BYTE;
	pos: INT;
END_VAR

(*
version 1.1	29. mar. 2008
programmer 		kurt
tested by		hugo

IS_UPPER testet ob in einem string keine Kleinbuchstaben vorkommen.

*)

PT := ADR(str);
L := LEN(str);
FOR pos := 1 TO L DO
	IF NOT (ISC_UPPER(pt^)) THEN
		IS_UPPER := FALSE;
		RETURN;
	END_IF;
    	PT := PT + 1;
END_FOR;
IS_UPPER := L > 0;


(* revision history
hm	29. feb 2008	rev 1.0
	original version

hm	29. mar. 2008	rev 1.1
	changed STRING to STRING(STRING_LENGTH)
*)

END_FUNCTION

// oscat_basic/POUs/String/ISC_UPPER
FUNCTION ISC_UPPER : BOOL
VAR_INPUT
	IN : BYTE;
END_VAR


(*
version 1.1	19. oct. 2008
programmer 	hugo
tested by	oscat

ISC_upper checks if a character is uppercase

*)

IF setup.EXTENDED_ASCII THEN
	ISC_UPPER :=  ((in > 64) AND (in < 91)) OR (((in > 191) AND (in < 223)) AND (in <> 215));
ELSE
	ISC_UPPER := ((in > 64) AND (in < 91));
END_IF;


(* revision history
hm	6. mar. 2008	rev 1.0
	original version

hm	19. oct. 2008	rev 1.1
	changes setup constants

*)

END_FUNCTION

// oscat_basic/POUs/String/MESSAGE_4R
FUNCTION_BLOCK MESSAGE_4R
VAR_INPUT
	M0 : STRING(STRING_LENGTH);
	M1 : STRING(STRING_LENGTH);
	M2 : STRING(STRING_LENGTH);
	M3 : STRING(STRING_LENGTH);
	MM : INT := 3;
	ENQ : BOOL := TRUE;
	CLK : BOOL := TRUE;
	T1 : TIME := T#3s;
END_VAR
VAR_OUTPUT
	MX : STRING(STRING_LENGTH);
	MN : INT;
	TR : BOOL;
END_VAR
VAR
	timer : TON;
	edge: BOOL;
END_VAR

(*
version 1.1	27. oct. 2008
programmer 	hugo
tested by	tobias

this function generates a rotation meassage with up to 4 strings.
on each rising edge of EN the next message in line will be displayed.
when EN stays high longer then one cycle, the next message will be displayed automatically after the time T1 is elapsed.
the output MX is the generated message and CX is a counter 0..3 signaling the current message displayed.
the displayed messages are 0 .. MM.

*)

(* check for rising edge on EN *)
TR := FALSE;
IF ENQ THEN
	IF (NOT edge AND clk) OR timer.q THEN
			MN := INC1(MN, MM);
			TR := TRUE;
			timer(in := FALSE);
			CASE MN OF
				0 : MX := M0;
				1 : MX := M1;
				2 : MX := M2;
				3 : MX := M3;
			END_CASE;
	END_IF;
	edge := clk;
	timer( in := CLK, pt := T1);
ELSE
	MX := '';
	MN := 0;
END_IF;




(* revision history
hm	8. oct. 2008	rev 1.0
	original version

hm	27. oct. 2008	rev 1.1
	changed _INC to INC1

*)

END_FUNCTION_BLOCK

// oscat_basic/POUs/String/MESSAGE_8
FUNCTION_BLOCK MESSAGE_8
VAR_INPUT
	IN1 : BOOL;
	IN2 : BOOL;
	IN3 : BOOL;
	IN4 : BOOL;
	IN5 : BOOL;
	IN6 : BOOL;
	IN7 : BOOL;
	IN8 : BOOL;
END_VAR
VAR_INPUT CONSTANT
	S1 : STRING(STRING_LENGTH);
	S2 : STRING(STRING_LENGTH);
	S3 : STRING(STRING_LENGTH);
	S4 : STRING(STRING_LENGTH);
	S5 : STRING(STRING_LENGTH);
	S6 : STRING(STRING_LENGTH);
	S7 : STRING(STRING_LENGTH);
	S8 : STRING(STRING_LENGTH);
END_VAR
VAR_OUTPUT
	M : STRING(STRING_LENGTH);
END_VAR


(*
version 1.1	29. mar. 2008
programmer 	hugo
tested by	tobias

this function generates one out of 4 messages specified by S1 .. S8.
the selected message will be presented at the output M.
In1 has higher priority then In2 which has higher priority then IN3 and in8 has the lowest priority.
*)

(* check if an alarm is present if yes set the output M otherwise clear M *)
IF in1 THEN
	M := S1;
ELSIF in2 THEN
	M := S2;
ELSIF in3 THEN
	M := S3;
ELSIF in4 THEN
	M := S4;
ELSIF in5 THEN
	M := S5;
ELSIF in6 THEN
	M := S6;
ELSIF in7 THEN
	M := S7;
ELSIF in8 THEN
	M := S8;
ELSE
	M := '';
END_IF;

(* revision history
hm	26.12.2007		rev 1.0
	original version

hm	29. mar. 2008	rev 1.1
	changed STRING to STRING(STRING_LENGTH)
*)

END_FUNCTION_BLOCK

// oscat_basic/POUs/String/MIRROR
FUNCTION MIRROR : STRING(STRING_LENGTH)
VAR_INPUT
	str : STRING(STRING_LENGTH);
END_VAR
VAR
	pi : POINTER TO ARRAY[1..255] OF BYTE;
	po : POINTER TO BYTE;
	lx: INT;
	i: INT;
END_VAR

(*
version 1.1	29. mar. 2008
programmer 	hugo
tested by	tobias

this function reverses an input string.

*)

pi := ADR(str);
po := ADR(mirror);
lx := LEN(str);
FOR i := lx TO 1 BY - 1 DO
	po^ := pi^[i];
	po := po + 1;
END_FOR;
(* close output string *)
po^:= 0;


(* revision histroy
hm	4. feb. 2008	rev 1.0
	original release

hm	29. mar. 2008	rev 1.1
	changed STRING to STRING(STRING_LENGTH)
*)

END_FUNCTION

// oscat_basic/POUs/String/REAL_TO_STRF
FUNCTION REAL_TO_STRF : STRING(20)
VAR_INPUT
	IN : REAL;
	N : INT;
	D : STRING(1);
END_VAR
VAR
	O: REAL;
	i: INT;
END_VAR

(*
version 1.8	2. jan 2012
programmer 	hugo
tested by	oscat

Real_to_strf converts a Real to a fixed length String.
the string will be filles with zeroes to achieve the fixed length N after the decimal separator.
the input parameter specifies the decimal separator to be used in the output string.

*)

(* LIMIT N to 0 .. 7 *)
N := LIMIT(0,N,7);
(* round the input to N digits and convert to string *)
O := ABS(in) * EXP10(N);
REAL_TO_STRF := DINT_TO_STRING(REAL_TO_DINT(O));
(* add zeroes in front to make sure sting is at least 8 digits long *)
FOR i := LEN(REAL_TO_STRF) TO N DO REAL_TO_STRF := CONCAT('0', REAL_TO_STRF); END_FOR;
(* add a dot if n > 0 *)
IF n > 0 THEN REAL_TO_STRF := INSERT(REAL_TO_STRF, D, LEN(REAL_TO_STRF) - N); END_IF;
(* add a minus sign if in is negative *)
IF in < 0 THEN REAL_TO_STRF := CONCAT('-', REAL_TO_STRF); END_IF;


(* revision history
hm	26 jan 2007	rev 1.0
	original version

hm	20. nov. 2007	rev 1.1
	when N=0 ther will be no dot at the end of the string.

hm	15. dec. 2007	rev 1.2
	changed code for better performance

hm	4. mar. 2008	rev 1.3
	result is now rounded instead of trunc

hm	20. mar. 2008	rev 1.4
	changed trunc to real_to_dint because trunc was generating wrong values on wago 842

hm	29. mar. 2008	rev 1.5
	changed STRING to STRING(20)

hm	4. apr. 2008	rev 1.6
	added variable O to avoid an error uner CoDeSys SP PLCWinNT V2.4

hm	27. feb. 2009	rev 1.7
	added a missing zero for IN < 1

hm 2. jan 2012	rev 1.8
	added input parameter D to specify decimal separator
*)

END_FUNCTION

// oscat_basic/POUs/String/REPLACE_ALL
FUNCTION REPLACE_ALL : STRING(STRING_LENGTH)
VAR_INPUT
	str : STRING(STRING_LENGTH);
	src : STRING(STRING_LENGTH);
	rep : STRING(STRING_LENGTH);
END_VAR
VAR
	pos: INT;
	lp : INT;
	lx : INT;
END_VAR

(*
version 1.1	29. mar. 2008
programmer 	hugo
tested by	tobias

the function replace_all replaces all occurences of src in str and replaces them by rep.

*)

REPLACE_ALL := str;
lx := LEN(src);
lp := LEN(rep);
pos := FINDP(REPLACE_ALL, src, 1);
WHILE pos > 0 DO
	REPLACE_ALL := REPLACE(REPLACE_ALL,rep,lx, pos);
	pos := FINDP(REPLACE_ALL, src, pos + lp);
END_WHILE;

(* revision histroy
hm	4. feb. 2008	rev 1.0
	original release

hm	29. mar. 2008	rev 1.1
	changed STRING to STRING(STRING_LENGTH)
*)

END_FUNCTION

// oscat_basic/POUs/String/REPLACE_CHARS
FUNCTION REPLACE_CHARS : STRING(STRING_LENGTH)
VAR_INPUT
	STR : STRING(STRING_LENGTH);
	SRC : STRING;
	REP : STRING;
END_VAR
VAR
	a, b : INT;
	c: STRING(1);
	stp: INT;
END_VAR

(*
version 1.0		14. may. 2008
programmer 		hugo
tested by			hugo

REPLACE_CHARS erstezt alle character die im string src aufgeführt sind mit dem an der selben stelle im string rep gelisteten character.

*)

REPLACE_CHARS := STR;
(* make sure rep and src are of same length and length is > 0 *)
a := LEN(src);
b := LEN(rep);
IF a < b THEN
	rep := LEFT(rep, a);
ELSIF b < a THEN
	src := LEFT(src, b);
END_IF;

(* search the string and replace if necessary *)
stp := LEN(str);
FOR a := 1 TO stp DO
	c := MID(REPLACE_CHARS, 1, a);
	b := FIND(src, c);
	IF b > 0 THEN
		REPLACE_CHARS := REPLACE(REPLACE_CHARS, MID(rep, 1, b), 1, a);
	END_IF;
END_FOR;



(* revision history
hm	14. may. 2008	rev 1.0
	original version

*)

END_FUNCTION

// oscat_basic/POUs/String/REPLACE_UML
FUNCTION REPLACE_UML : STRING(STRING_LENGTH)
VAR_INPUT
	str : STRING(STRING_LENGTH);
END_VAR
VAR
	L : INT;
	pt : POINTER TO BYTE;
	pto : POINTER TO BYTE;
	ptm : POINTER TO BYTE;
	pt1, pt2 : POINTER TO BYTE;
	su : STRING(2);
	pos : INT;
END_VAR

(*
version 1.1	29. mar. 2008
programmer 		kurt
tested by		hugo

REPLACE_UML replaces all occurences of Ä,Ö,Ü and ä,ö,ü,ß with Ae, ae, Oe, oe, Ue, ue and ss.

*)

PT := ADR(str);
pto := ADR(REPLACE_UML);
ptm := pto + INT_TO_DWORD(string_length);
pt1 := ADR(su);
pt2 := pt1 + 1;
L := LEN(str);
WHILE pos < L AND pos < string_length DO
	IF pt^ < 127 THEN
		(* no uml character simlply copy the character*)
		pto^ := pt^;
	ELSE
		(* convert the uml character *)
		su := TO_UML(pt^);
		(* we must make sure pointer are not out of range *)
		pto^ := pt1^;
		IF pto < ptm AND pt2^ > 0 THEN
			pto := pto + 1;
			pto^ := pt2^;
		END_IF;
	END_IF;
	(* increment pointers *)
	pt := pt + 1;
	pto := pto + 1;
	pos := pos + 1;
END_WHILE;

(* properly close the output string *)
pto^ := 0;


(* revision history
hm	29. feb 2008	rev 1.0
	original version

hm	29. mar. 2008	rev 1.1
	changed STRING to STRING(STRING_LENGTH)
	new code to avoid pointer out of range
	use new function to_uml
*)

END_FUNCTION

// oscat_basic/POUs/String/TO_UML
FUNCTION TO_UML : STRING(2)
VAR_INPUT
	IN : BYTE;
END_VAR


(*
version 1.1	17. dec. 2008
programmer 		hugo
tested by		tobias

to_uml converts a character above 127 to a two digit character below 127.
the character Ä is converted to Ae

*)

CASE in OF
	196:	(* Ä *)
		TO_UML := 'Ae';
	214:	(* Ö *)
		TO_UML := 'Oe';
	220:	(* Ü *)
		TO_UML := 'Ue';
	223:	(* ß *)
		TO_UML := 'ss';
	228:	(* ä *)
		TO_UML := 'ae';
	246:	(* ö *)
		TO_UML := 'oe';
	252:	(* ü *)
		TO_UML := 'ue';
ELSE
	TO_UML := CHR_TO_STRING(IN);
END_CASE;



(* revision history
hm	29. mar. 2008	rev 1.0
	original version

hm	17. dec. 2008	rev 1.1
	changes name of function chr to chr_to_string

*)

END_FUNCTION

// oscat_basic/POUs/String/TICKER
FUNCTION_BLOCK TICKER

VAR_INPUT
	N : INT;
	PT : TIME;
END_VAR

VAR_INPUT
	Text : STRING(STRING_LENGTH);
END_VAR

VAR_OUTPUT
	Display : STRING(STRING_LENGTH);
END_VAR
VAR
	delay : TP;
	step : INT;
END_VAR

(*
version 1.2	29. mar. 2008
programmer 	hugo
tested by		tobias

Ticker sends a substring of text with length N every TD Milliseconds to generate a ticker. 

*)


(* generate next ticker when delay is low *)
IF N < LEN(text) THEN
	IF NOT delay.Q THEN
		(* increase step for next tick *)
		step := step + 1;
		IF step > LEN(text) THEN step := 1; END_IF;
		(* extract dispay from text *)
		display := MID(text, N, step);
		(* set delay timer for next tick *)
		delay(in := TRUE, PT := PT);
	ELSE;
		(* execute delay timer *)
		delay(in := FALSE);
	END_IF;
ELSE
	display := text;
END_IF;
(* revision history
hm	4. dec. 2007	rev 1.0
	original version

hm	15. dec. 2007	rev 1.1
	step now starts at 1 instaed of 0

hm	29. mar. 2008	rev 1.2
	changed STRING to STRING(STRING_LENGTH)
*)

END_FUNCTION_BLOCK

// oscat_basic/POUs/String/TRIM1
FUNCTION TRIM1 : STRING(STRING_LENGTH)
VAR_INPUT
	str : STRING(STRING_LENGTH);
END_VAR
VAR
	pos: INT;
END_VAR

(*
version 1.2	29. mar. 2008
programmer 	hugo
tested by		tobias

the function replaces all multiple blanks within a string by only one blank.
leading and ending blanks will be deleted

*)

TRIM1 := str;
REPEAT
	pos := FIND(trim1,'  ');
	IF pos > 0 THEN TRIM1 := REPLACE(TRIM1,' ',2,pos); END_IF;
UNTIL pos = 0	END_REPEAT;
(* beginning and ending blanks need to be stripped off *)
IF LEFT(trim1,1) = ' ' THEN trim1 := DELETE(trim1,1,1); END_IF;
IF RIGHT(trim1,1) = ' ' THEN trim1 := DELETE(trim1,1,LEN(trim1)); END_IF;


(* revision histroy
hm	4. feb. 2008    rev 1.0
	original release

hm	20. mar. 2008	rev 1.1
	avoid to call replace with pos = 0 because some systems will produce an error

hm	29. mar. 2008	rev 1.2
	changed STRING to STRING(STRING_LENGTH)
*)

END_FUNCTION

// oscat_basic/POUs/String/TRIME
FUNCTION TRIME : STRING(string_length)
VAR_INPUT
	str : STRING(STRING_LENGTH);
END_VAR


(*
version 1.0	28. mar. 2008
programmer 	hugo
tested by	tobias

this function deletes all leading and ending blanks of a string.

*)

TRIME := str;
(* beginning blanks need to be stripped off *)
WHILE LEFT(TRIME,1) = ' ' DO
	TRIME := DELETE(TRIME,1,1);
END_WHILE;

(* ending blanks need to be stripped off *)
WHILE RIGHT(TRIME,1) = ' ' DO
	TRIME := DELETE(TRIME,1,LEN(TRIME));
END_WHILE;


(* revision histroy
hm	28. mar. 2008	rev 1.0
	original release

*)

END_FUNCTION

// oscat_basic/POUs/Time&Date/CALENDAR_CALC
FUNCTION_BLOCK CALENDAR_CALC
VAR_INPUT
	SPE : BOOL;
	H : REAL := -0.83333333333;
END_VAR
VAR_IN_OUT
	XCAL : CALENDAR;
	HOLIDAYS : ARRAY[0..29] OF HOLIDAY_DATA;
END_VAR
VAR
	last : DT;
	last_day : DINT;
	holy : HOLIDAY;
	sun : SUN_TIME;
	last_hour: INT;
	utod: TOD;
	pos : SUN_POS;
	plast: DT;
END_VAR
VAR
	dtemp : DINT;
	tmp : INT;
END_VAR


(*
version 1.6	6. apr. 2011
programmer 	hugo
tested by		oscat

calendar_calc liest die weltzeit .UTC aus einer CALENDAR Struktur und berechnet die restlichen Werte der Struktur.
calendar_calc stellt sicher das die Werte fortlaufend aktualisiert werden und dabei funktionen nur dann aufgerufen werden wenn dies nötig ist.
calendar_calc will calculate sun position data when SPE = TRUE;

*)

IF xcal.UTC <> last THEN
	(* run once per second *)
	(* update utc last calculated  *)
	last := XCAL.UTC;
	utod := DT_TO_TOD(xcal.UTC);

	(* calculate ltc from utc *)
	XCAL.LDT := UTC_TO_LTIME(XCAL.UTC, XCAL.DST_EN, XCAL.OFFSET);
	XCAL.LDATE := DT_TO_DATE(XCAL.LDT);
	XCAL.LTOD := DT_TO_TOD(XCAL.LDT);
	dtemp := DAY_OF_DATE(XCAL.LDATE);
	xcal.night := XCAL.LTOD < XCAL.SUN_RISE OR XCAL.LTOD > XCAL.SUN_SET;

	(* run once per hour *)
	tmp := HOUR(xcal.LTOD);
	IF  tmp <> last_hour THEN
		XCAL.DST_ON := DST(XCAL.UTC) AND xcal.DST_EN;
		last_hour := tmp;
	END_IF;

	(* run once per day *)
	IF dtemp <> last_day THEN
		last_day := dtemp;
		(* a new day has started, recalculate daily events *)
		XCAL.YEAR := YEAR_OF_DATE(XCAL.LDATE);
		XCAL.MONTH := MONTH_OF_DATE(XCAL.LDATE);
		XCAL.DAY := DAY_OF_MONTH(XCAL.LDATE);
		XCAL.WEEKDAY := DAY_OF_WEEK(XCAL.LDATE);
		HOLY(date_in := XCAL.LDATE, LANGU := xcal.LANGUAGE, HOLIDAYS := HOLIDAYS);
		XCAL.HOLIDAY := HOLY.Y;
		XCAL.HOLY_NAME := HOLY.NAME;
		sun(latitude := XCAL.LATITUDE, longitude := xcal.LONGITUDE, utc := DT_TO_DATE(xcal.UTC), H := H);
		XCAL.SUN_RISE := DINT_TO_TOD(TOD_TO_DINT(sun.sun_rise) + XCAL.OFFSET * 60000 + SEL(XCAL.DST_ON,DINT#0,3600000));
		XCAL.SUN_SET := DINT_TO_TOD(TOD_TO_DINT(sun.sun_set) + XCAL.OFFSET * 60000 + SEL(XCAL.DST_ON,DINT#0,3600000));
		XCAL.SUN_MIDDAY := DINT_TO_TOD(TOD_TO_DINT(sun.MIDDAY) + XCAL.OFFSET * 60000 + SEL(XCAL.DST_ON,DINT#0,3600000));
		XCAL.SUN_HEIGTH := sun.sun_declination;
		XCAL.WORK_WEEK := WORK_WEEK(XCAL.LDATE);
	END_IF;

	(* calculate the suns position every 10 seconds when SPE = TRUE *)
	IF SPE AND xcal.UTC -  plast >= t#25s THEN
		plast := last;
		pos(latitude := xcal.LATITUDE, longitude := xcal.LONGITUDE, utc := xcal.UTC);
		xcal.SUN_HOR := pos.B;
		xcal.SUN_VER := pos.HR;
	END_IF;
END_IF;



(* revision history

hm 23. oct. 2008	rev 1.0
	original version

hm	8. feb. 2009	rev 1.1
	night was calculated wrong
	added sun position data

hm	10. mar. 2009	rev 1.2
	added work_week, sun_midday, sun_heigth
	sun_position will only be calculated evey 25 seconds
	dst will only become true when dst_en = true

hm	23. jan 2010	rev 1.3
	sun_rise, sun_set and sun_midday are now calculated in local time

hm	18. jan. 2011	rev 1.4
	added input holidays to specify local holidays
	changed call for function sun_time

hm	2. feb. 2011	rev 1.5
	added input H to specify twilight

hm	6. apr. 2011	rev 1.6
	night was calculated wrong
*)

END_FUNCTION_BLOCK

// oscat_basic/POUs/Time&Date/UTC_TO_LTIME
FUNCTION UTC_TO_LTIME : DT
VAR_INPUT
	UTC : DT;
	DST_ENABLE : BOOL;
	TIME_ZONE_OFFSET : INT;
END_VAR
VAR
	tmp: INT;
END_VAR

(*

version 1.9	27. feb. 2009
programmer 	oscat
tested by		oscat

ltime is a real time clock that uses the system rtc as utc time and calculates and given time zone.
the utc time is supplied on the input UTC.
according to the input variable time_zone_offset when the input dst_enable is true,
the dst on and off times are calculated by a formula for any given year and the time is advanced and reset by one hour
at 02:00 and 03:00 for the last sunday of march and last sunday of october.
the code is high performance and the rtc counts every second.
if more then one time zone is needed by the systen the clock can be started many times by placing more then one function block.

 
*)

tmp := TIME_ZONE_OFFSET * 60 + BOOL_TO_INT(DST_ENABLE AND DST(UTC)) * 3600;
IF tmp < 0 THEN
	tmp := ABS(tmp);
	UTC_TO_LTIME := DWORD_TO_DT(DT_TO_DWORD(UTC) -  INT_TO_DWORD(tmp));
ELSE
	UTC_TO_LTIME := DWORD_TO_DT(DT_TO_DWORD(UTC) +  INT_TO_DWORD(tmp));
END_IF;


(* revision history

hm 2.10.2006	rev 1.1
	corrected an error where dst would be delayed by 0.1second

hm 17.1.2007	rev 1.2
	added utc input instead of internal sysrtcgettime because this would only work on wago.
	dst_enable would not be checked before dst would be enabled.

hm 18.3.2007	rev 1.3
	changed code, dst would not work during first cycle.

hm 24.10.2007	rev 1.4
	changed code because the execution every 100ms can cause major problems if the supplied time was not correct at start.
	use of new dst function

hm 12. nov 2007	rev 1.5
		changed Type of time_zone_offset from time to int to allow for time zones with negative offset

hm	8 dec 2007		rev 1.6
	corrected a problem with time_zone_offset

hm	14. oct. 2008	rev 1.7
	renamed module from LTIME to UTC_TO_LTIME
	changed function weekday to day_of_week
	optimized code for better performance

hm	20. oct. 2008	rev 1.8
	changes type of input TIME_ZONE_OFFSET from real to int, now is in +/-minutes
	deleted outputs DST_ON and WDAY
	converted to function

hm	27. feb. 2009	rev 1.9
	added type conversions to avoid warnings under codesys 3.0

*)

END_FUNCTION

// oscat_basic/POUs/Time&Date/DST
FUNCTION DST : BOOL
VAR_INPUT
	UTC : DT;
END_VAR
VAR
	yr : INT;
	yr4 : DWORD;
	ltc: DWORD;
	idate : DWORD;
END_VAR

(*
version 1.5	24. jan. 2011
programmer 	hugo
tested by	oscat

this functions returns TRUE IF dst TIME is active 
the FUNCTION calculates automatically for any year betweek 1970 AND 2099 
wheather daylight savings is on OR off 
the summertime calculation is done according to european standards.
dst will become TRUE AT 01:00 utc in the morning FOR the respective days 
AND it will become FALSE after daylight savings TIME is switched back end OF october at 01:00 utc

*)

yr := YEAR_OF_DATE(DT_TO_DATE(UTC));
ltc := DT_TO_DWORD(UTC);
idate := DT_TO_DWORD(SET_DT(yr, 3, 31, 1, 0, 0));
yr4 := SHR(5 * INT_TO_DWORD(yr), 2) + 1;
DST := (idate - ((yr4 + 3) MOD 7) * 86400 <= ltc) AND (idate + (214 - (yr4) MOD 7) * 86400 > ltc);


(*
Equation used TO calculate the beginning OF European Summer TIME:
Sunday (31 - (5*y/4 + 4) mod 7) March at 01.00 UTC
(valid through 2099, courtesy of Robert H. van Gent, EC).

European Summer Time ends (clocks go back) at 01.00 UTC on

    * 29 October 2006
    * 28 October 2007
    * 26 October 2008

Equation used to calculate the end of European Summer Time:
Sunday (31 - (5*y/4 + 1) mod 7) October at 01.00 UTC
(validity AND credits as above).

*)



(* revision history
hm	4. aug 2006	rev 1.0
	original version

hm	24. okt 2007	rev 1.1
	deleted time_zone_offset input because dst is generally at 01:00 utc and not mesz
	uk starts 01:00 utc and also greece

hm	1. dec 2007	rev 1.2
	changed code to improve performance

hm	16. mar. 2008	rev 1.3
	added type conversion to avoid warnings under codesys 3.0
	code improvement for better performance

hm	7. oct. 2008	rev 1.4
	changed name of function year to year_of_date

hm	24. jan. 2011	rev 1.5
	improved performance
*)

END_FUNCTION

// oscat_basic/POUs/Time&Date/HOLIDAY
FUNCTION_BLOCK HOLIDAY
VAR_INPUT
	DATE_IN : DATE;
	LANGU : INT;
	FRIDAY : BOOL;
	SATURDAY : BOOL;
	SUNDAY : BOOL;
END_VAR
VAR_IN_OUT
	HOLIDAYS : ARRAY[0..29] OF HOLIDAY_DATA;
END_VAR
VAR CONSTANT
	SIZE : INT := 29;
END_VAR
VAR_OUTPUT
	Y : BOOL;
	NAME : STRING(30);
END_VAR
VAR
	last_active : DATE;
	ostern: DATE;
	i: INT;
	jahr: INT;
	x_date: DATE;
	lx: INT;
	wdx: INT;
END_VAR

(*
version 2.0	18. jans 2011
programmer 	hugo
tested by		tobias

holiday calculates if a given day is a holiday and displays the name of the holiday as string as well as a boolean flag to indicate a holiday.
the holidays are specified in the country setup under global constants.
a holiday can be of fixed date for example new years day on january 1st.
a holiday can have a fixed offset from easter sunday as for most church holidays.
a holiday can be a specific weekday before a fixed date, for example buss und bettag is the last wednesday before nov 23rd.
with a simple f_use flag any specific holiday can be turned on or off if needed.

please check the manual for examples of holiday definitions
*)

(* for performance reasons only activate once a day *)
IF last_active = date_in THEN RETURN; END_IF;
last_active := DATE_IN;

(* determine language *)
IF LANGU = 0 THEN
	lx := language.DEFAULT;
ELSE
	lx := MIN(language.LMAX, LANGU);
END_IF;

(* berechnung von ostern für das aktuelle jahr *)
jahr := YEAR_OF_DATE(date_in);
ostern := EASTER(jahr);
wdx := DAY_OF_WEEK(DATE_IN);
Y := FALSE;

(* check for holidays *)
FOR i := 0 TO size DO
	x_date := SET_DATE(jahr, HOLIDAYS[i].MONTH , HOLIDAYS[i].DAY);
	IF HOLIDAYS[i].USE = 1 AND HOLIDAYS[i].MONTH > 0 THEN
		(* check for fixed date holiday *)
		IF x_date = date_in THEN
			Y := TRUE;
			NAME := HOLIDAYS[i].NAME;
			RETURN;
		END_IF;
	ELSIF HOLIDAYS[i].USE = 1 AND HOLIDAYS[i].MONTH = 0 THEN
		(* check for holiday in reference to easter *)
		IF DATE_ADD(ostern, HOLIDAYS[i].DAY ,0,0,0) = date_in THEN
			Y := TRUE;
			NAME := HOLIDAYS[i].NAME;
			RETURN;
		END_IF;
	ELSIF HOLIDAYS[i].USE < 0 THEN
		(* check for holiday on a weekday before date *)
		IF DAY_OF_WEEK(date_in) = ABS(HOLIDAYS[i].USE) AND date_in < x_date AND date_in >= DATE_ADD(x_date,-7,0,0,0) THEN
			Y := TRUE;
			NAME := HOLIDAYS[i].NAME;
			RETURN;
		END_IF;
	END_IF;
END_FOR;

(* check array if today is weekend *)
IF NOT Y AND (wdx = 5 AND FRIDAY OR wdx = 6 AND SATURDAY OR wdx = 7 AND SUNDAY) THEN
	Y := TRUE;
	NAME := LANGUAGE.WEEKDAYS[LOCATION.LANGUAGE[lx],wdx];
ELSE
	NAME := '';
END_IF;


(*
Neujahrstag 	1. Januar 	• 	• 	• 	• 	• 	• 	• 	• 	• 	• 	• 	• 	• 	• 	• 	•
Heilige Drei Könige 	6. Januar 	• 	• 												• 		
Karfreitag 	Ostersonntag - 2d 	• 	• 	• 	• 	• 	• 	• 	• 	• 	• 	• 	• 	• 	• 	• 	•
Ostersonntag 	siehe Osterdatum 				(•) 												
Ostermontag 	Ostersonntag + 1d 	• 	• 	• 	• 	• 	• 	• 	• 	• 	• 	• 	• 	• 	• 	• 	•
Tag der Arbeit 	1. Mai 	• 	• 	• 	• 	• 	• 	• 	• 	• 	• 	• 	• 	• 	• 	• 	•
Christi Himmelfahrt 	Ostersonntag + 39d 	• 	• 	• 	• 	• 	• 	• 	• 	• 	• 	• 	• 	• 	• 	• 	•
Pfingstsonntag 	Ostersonntag + 49d 				(•) 												
Pfingstmontag 	Ostersonntag + 50d 	• 	• 	• 	• 	• 	• 	• 	• 	• 	• 	• 	• 	• 	• 	• 	•
Fronleichnam 	Ostersonntag + 60d 	• 	• 					• 			• 	• 	• 	1) 			2)
Augsburger Friedensfest 	8. August 		(3) 														
Mariä Himmelfahrt 	15. August 		(5) 										• 				
Tag der Deutschen Einheit 	3. Oktober 6) 	• 	• 	• 	• 	• 	• 	• 	• 	• 	• 	• 	• 	• 	• 	• 	•
Reformationstag 	31. Oktober 				• 				• 					• 	• 		•
Allerheiligen 	1. November 	• 	• 								• 	• 	• 				
Buß- und Bettag 4) 	Mittwoch vor dem 23.11. 			7 										• 			
1. Weihnachtstag 	25. Dezember 	• 	• 	• 	• 	• 	• 	• 	• 	• 	• 	• 	• 	• 	• 	• 	•
2. Weihnachtstag 	26. Dezember 	• 	• 	• 	• 	• 	• 	• 	• 	• 	• 	• 	• 	• 	• 	• 	•
*)



(* revision history
hm 	27. feb. 2007	rev 1.1
	deleted unused variable init

hm	31. oct. 2007	rev 1.2
	changed holiday definition from constant to input constant to allow easier changes by user without recompilation of the lib

hm 	24. nov. 2007	rev 1.3
	changes F_use of  Buß_und_Bettag to 0 because this is no official holiday

hm	7. apr. 2008	rev 1.4
	improved performance

hm	7. oct. 2008	rev 1.5
	changed code to use setup data from global constants
	changed length of output NAME from 20 to 30
	holiday will now also be indicated on a weekend
	changed function year to year_of_date
	changed function weekday to day_of_week

hm	21. oct. 2008	rev 1.6
	using location constants

hm	18. jan 2011	rev 2.0
	using user specified array for holidays

*)

END_FUNCTION_BLOCK

// oscat_basic/POUs/Time&Date/EASTER
FUNCTION EASTER : DATE
VAR_INPUT
	year : INT;
END_VAR
VAR
	b,c: INT;
	oday: INT;
END_VAR

(*
version 1.3	7. apr. 2008
programmer 	hugo
tested by	tobias

easter calculates the day of easter sunday for a given year.
most other catholic holidays are calculated in reference to easter sunday.

*)

b := (204 - 11 * (YEAR MOD 19)) MOD 30;
IF b > 27 THEN b := b - 1; END_IF;
c := (year + SHR(year,2) + b - 13) MOD 7;
oday := 28 + b - c;
IF oday > 33 THEN
	EASTER := SET_DATE(year, 4, oday - 31);
ELSE
	EASTER := SET_DATE(year, 3, oday);
END_IF;




(* alternativer algorithmus ueber das pasah fest
execution time roughly 200us
Der sog. Passah-Vollmond wird berechnet, in dem das Jahr durch 19 ge-
teilt wird und der Rest mit der folgenden Tabelle verglichen wird:
 
    0: Apr 14       5: Apr 18      10: Mrz 25      15: Mrz 30
    1: Apr 03       6: Apr 08      11: Apr 13      16: Apr 17
    2: Mrz 23       7: Mrz 28      12: Apr 02      17: Apr 07
    3: Apr 11       8: Apr 16      13: Mrz 22      18: Mrz 27
    4: Mrz 31       9: Apr 05      14: Apr 10
 
Faellt dieses Datum auf einen Sonntag, ist Ostern der naechste Sonntag!
 
Beispiel: 1992 MOD 19 = 16, daraus folgt 17.04., der naechste Sonntag
          ist dann der 19. April (Ostersonntag)
*)


(* this algorithm is 180 us
a := year MOD 19;
b := year / 100;
c := year MOD 100;
d := b / 4;
e := b MOD 4;
f := (b + 8) / 25;
g := (b - f + 1) / 3;
h := (19 * a + b - d -g + 15) MOD 30;
i := C / 4;
k := c MOD 4;
l := (32 + 2*e + 2*i - h - k) MOD 7;
m := (a + 11 * h + 22 * l) / 451;
x := h + l - 7 * m + 114;
n := X / 31;
o := x MOD 31 + 1;

easter := set_Date(year,n,o);
*)
(*
Im Magazin "Nature" vom 20. April 1876 veröffentlichte ein anonymer Autor eine Tabelle mit Regeln zur Berechnung des (Gregorianischen) Ostersonntages des Jahres J. In Formeln ausgedrückt erhält man das Folgende:
a	=	J mod 19
b	=	int(J / 100)
c	=	J mod 100
d	=	int(b / 4)
e	=	b mod 4
f	=	int((b + 8) / 25)
g	=	int((b - f + 1) / 3
h	=	(19 · a + b - d - g + 15) mod 30
i	=	int(c / 4)
k	=	c mod 4
l	=	(32 + 2 · e + 2 · i - h - k) mod 7
m	=	int((a + 11 · h + 22 · l) / 451)
n	=	int((h + l - 7 · m + 114) / 31)
o	=	(h + l - 7 · m + 114) mod 31

n ist hierbei die Nummer des Monats, o + 1 die Nummer des Tages auf welchen der Ostersonntag im Jahr J fällt. Dieser Algorithmus kommt ohne Hilfszahlen aus.

*)

(* revision history
hm	27. dec 2006	rev 1.0
	original version

hm	15. dec 2007	rev 1.1
	modified code for better performance

hm	3. feb 2008		rev 1.2
	modified code for better performance

hm	7. apr. 2008	rev 1.3
	improved performance
*)

END_FUNCTION

// oscat_basic/POUs/Time&Date/SUN_MIDDAY
FUNCTION SUN_MIDDAY : TOD
VAR_INPUT
	LON : REAL;
	UTC : DATE;
END_VAR
VAR
	T : REAL;
	OFFSET : REAL;
END_VAR

(*
version 1.0	26. jan. 2011
programmer 	hugo
tested by	oscat

this FUNCTION calculates the time when the sun stand exactly south of a given location.

*)

T := INT_TO_REAL(DAY_OF_YEAR(utc));
OFFSET := -0.1752 * SIN(0.033430 * T + 0.5474) - 0.1340 * SIN(0.018234 * T - 0.1939);
SUN_MIDDAY := HOUR_TO_TOD(12.0 - OFFSET - lon * 0.0666666666666);


(* revision history

hm	26. jan. 2011	rev 1.0
	initial release

*)

END_FUNCTION

// oscat_basic/POUs/Time&Date/HOUR_TO_TOD
FUNCTION HOUR_TO_TOD : TOD
VAR_INPUT
	IN : REAL;
END_VAR


(*
version 1.2	24. feb 2009
programmer 	hugo
tested by		tobias

converts an amount of hours in real to time of day TOD.

*)

HOUR_TO_TOD := DWORD_TO_TOD(REAL_TO_DWORD(IN * 3600000));


(* revision history
hm	4. aug. 2006	rev 1.0
	original version

hm	14. mar. 2008	rev 1.1
	rounded the input after the last digit

hm	24. feb. 2009	rev 1.2
	changed input to IN
*)

END_FUNCTION

// oscat_basic/POUs/Time&Date/WORK_WEEK
FUNCTION WORK_WEEK : INT
VAR_INPUT
	idate : DATE;
END_VAR
VAR
	d1 : DATE;
	w1 : INT;
	ds: DWORD;
	yr: INT;
	w31: INT;
	w01: INT;
	wm: INT;
END_VAR

(*
version 1.5	25. oct. 2008
programmer 	hugo
tested by	oscat

calculates the work week for a given date according to iso8601

*)

(* berechne den 1.1 des jahres von idate. *)
yr := YEAR_OF_DATE(idate);
d1 := YEAR_BEGIN(yr);
(* wochentag von d1 *)
w1 := DAY_OF_WEEK(d1);
(* offset des montags der eletzten KW des vorjahres *)
(* wenn der erste tag des jahres größer als donnerstag ist dann beginnt die letzte kw am montag davor *)
(* wenn der erste tag des jahres ein donnerstag oder kleiner ist beginnt die erste kw 2 montage davor *)
IF w1 < 5 THEN
	ds := DATE_TO_DWORD(d1) - INT_TO_DWORD(w1+6) * 86400;
ELSE
	ds := DATE_TO_DWORD(d1) - INT_TO_DWORD(w1-1) * 86400;
END_IF;

(* kalenderwoche des eingangsdatums *)
WORK_WEEK := DWORD_TO_INT((DATE_TO_DWORD(idate) - ds) / 604800);

(* korrektur wenn work_week = 0 *)
IF work_week = 0 THEN
	(* work_week needs to be 53 when 1.jan of the year before is thursday or dec 31. is thursday. *)
	(* first and last weekday of a year is equal and one more day for a leap_year. *)
	IF w1 > 1 THEN w31 := w1 - 1; ELSE W31 := 7; END_IF;
	IF LEAP_YEAR(yr - 1) AND w31 > 1 THEN w01 := W31 - 1; ELSE w1 := 7; END_IF;
	(* if first or last day of a year is a thursday, the year has 53 weeks *)
	WORK_WEEK := 52 + BOOL_TO_INT(w31 = 4 OR w01 = 4);
ELSE
	(* end of year calculation *)
	(* calculated the first and last weekday *)
	IF leap_year(yr) THEN
		IF w1 < 7 THEN w31 := w1 + 1; ELSE w31 := 1; END_IF;
	ELSE
		w31 := w1;
	END_IF;
	(* if first or last day is thursday then the year has 53 weeks otherwise only 52 *)
	wm := 52 + BOOL_TO_INT(w31 = 4 OR w1 = 4);
	IF WORK_WEEK > wm THEN WORK_WEEK := 1; END_IF;
END_IF;



(* revision history

hm 	17.1.2007		rev 1.1
	deleted unused variable yday

hm	19. dec 2007	rev 1.2
	changed code for better performance
	changed code to comply with ISO8601

hm	16. mar 2008	rev 1.3
	added type conversions to avoid warnings under codesys 3.0

hm	7. oct. 2008	rev 1.4
	changed function year to year_of_date
	changed function weekday to day_of_week

hm	25. oct. 2008	rev 1.5
	optimized code for performance
*)

END_FUNCTION

// oscat_basic/POUs/Time&Date/SUN_TIME
FUNCTION_BLOCK SUN_TIME
VAR_INPUT
	LATITUDE : REAL;				(* latitude of geographical position  *)
	LONGITUDE : REAL;				(* longitude of geographical position  *)
	UTC : DATE;						(*	world time	*)
	H : REAL := -0.83333333333;	(* heighth above horizon for sunrise *)
END_VAR
VAR_OUTPUT
	MIDDAY : TOD;			(*	astrological midday in hours when sun stands at south direction	*)
	SUN_RISE : TOD;				(*	sun rise for current day in local time *)
	SUN_SET : TOD;				(*	sun set for current day in local time *)
	SUN_DECLINATION : REAL;		(*	sun declination above horizon at midday in degrees	*)
END_VAR
VAR
	dk: REAL;						(* sun declination at midday *)
	delta: TIME;					(* delta from midday for sunrise and sunset  *)
	b: REAL;
END_VAR

(*
version 1.7	25. jan. 2011
programmer 	hugo
tested by	tobias

this FUNCTION block calculates the sun rise, sun set, sun offset at midday sun declination for a given date 
for performance reasons the algorithm has been simplified and is accurate within a few minutes only 
the times are calculated in utc and have to be corrected for the given time zone
this correction is not done within sun_time because it would be a problem on days where dst is enabled or disabled

*)

B := latitude * 0.0174532925199433;
MIDDAY := SUN_MIDDAY(longitude, utc);
DK := 0.40954 * SIN(0.0172 * (INT_TO_REAL(DAY_OF_YEAR(utc)) - 79.35));
sun_declination := DEG(DK);
IF sun_declination > 180.0 THEN sun_declination := sun_declination - 360.0; END_IF;
sun_declination := 90.0 - LATITUDE + sun_declination;
delta := HOUR_TO_TIME(ACOS((SIN(RAD(H)) - SIN(B) * SIN(DK)) / (COS(B) * COS(DK))) * 3.819718632);
sun_rise := MIDDAY - delta;
sun_set := MIDDAY + delta;

(* revision history

rev 1.1	hm	20.1.2007
	deleted unused variables sun_riseR and sun_setR

rev 1.2 hm 17.4.2007
	corrected error while sun:midday would not be corrected for longitude.

rev 1.3	hm	6. jan 2008
	performance improvements

rev	1.4 hm	17. jan 2008
	calculation is now only performed once a day

hm	10. mar. 2009	rev 1.5
	improved performance
	calculation will be performed on every call to allow movong installations

hm	26. jul 2009	rev 1.6
	fixed a problem with wrong midday calculation

hm	25. jan. 2011	rev 1.7
	using function sun_midday
	corrected angle of sun_declination
	added input H
*)

END_FUNCTION_BLOCK

// oscat_basic/POUs/Time&Date/HOUR_TO_TIME
FUNCTION HOUR_TO_TIME : TIME
VAR_INPUT
	IN : REAL;
END_VAR


(*
version 1.2	24. feb. 2009
programmer 	hugo
tested by		tobias

converts an amount of hours in real to time

*)

HOUR_TO_TIME := DWORD_TO_TIME(REAL_TO_DWORD(IN * 3600000));


(* revision history
hm		4. aug 2006	rev 1.0
	original version

hm	14. mar. 2008	rev 1.1
	rounded the input after the last digit

hm	24. feb. 2009	rev 1.2
	changed input to IN
*)

END_FUNCTION

// oscat_basic/POUs/Time&Date/SUN_POS
FUNCTION_BLOCK SUN_POS
VAR_INPUT
	latitude : REAL;				(* latitude of geographical position  *)
	longitude : REAL;				(* longitude of geographical position  *)
	utc : DT;						(*	world time				*)
END_VAR
VAR_OUTPUT
	B: REAL;
	H : REAL;
	HR: REAL;
END_VAR
VAR
	g: REAL;
	a: REAL;
	d: REAL;
	t1: REAL;
	n: REAL;
	e: REAL;
	c: REAL;
	tau: REAL;
	sin_d: REAL;
	rlat: REAL;
	sin_lat: REAL;
	cos_lat: REAL;
	cos_tau: REAL;
	cos_d: REAL;
END_VAR

(*
version 2.1	7. mar. 2009
programmer 	hugo
tested by		oscat

this FUNCTION block calculates the sun position for a given date and time.
the times are calculated in utc and have to be corrected for the given time zone.
B is the angle from north and HR is the highth in degrees.

*)


(* n is the julian date and the number of days since 1.1.2000-12:00 midday *)
(* be careful for step7 date startes 1.1.1990 instead of 1.1.1970 *)
(* for step7 this line must change *)
n := DWORD_TO_REAL(DT_TO_DWORD(UTC) - 946728000) * 0.000011574074074074;
g :=MODR(6.240040768 + 0.01720197 * n, math.PI2);
d := MODR(4.89495042 + 0.017202792 * n, math.PI2) + 0.033423055 * SIN(g) + 0.000349066 * SIN(2.0*g);
e := 0.409087723 - 0.000000006981317008 * n;
cos_d := COS(d);
sin_d := SIN(d);
a := ATAN(COS(e) * sin_d / cos_d);
IF cos_d < 0.0 THEN a := a + math.PI; END_IF;
c := ASIN(SIN(e) * sin_d);

(* also here we must be very careful utc is from 1.1.1970 for step7 the formula must change *)
tau := RAD(MODR(6.697376 + (n - 0.25) * 0.0657098245037645 + DWORD_TO_REAL(TOD_TO_DWORD(DT_TO_TOD(utc))) * 0.0000002785383333, 24.0) * 15.0 + longitude) - a;
rlat := RAD(latitude);
sin_lat := SIN(rlat);
cos_lat := COS(rlat);
cos_tau := COS(tau);
t1 := cos_tau * sin_lat - TAN(c) * cos_lat;
B := ATAN(SIN(tau) / t1);
IF t1< 0.0 THEN B := B + math.PI2; ELSE B := B + math.PI; END_IF;
B := DEG(MODR(B, math.PI2));
h := DEG(ASIN(COS(C) * cos_tau * cos_lat +SIN(c) * sin_lat));
IF h > 180.0 THEN h := h - 360.0; END_IF;
(* consider refraction *)
HR := h + REFRACTION(h);


(* revision history
hm	1. feb 2007	rev 1.0
	original version

hm	6. jan 2008	rev 1.1
	performance improvements

hm	18. jan 2008	rev 1.2
	further performance improvements
	only calculate once every 10 seconds

hm	16. mar. 2008	rev 1.3
	added type conversion to avoid warnings under codesys 3.0

hm	30. jun. 2008	rev 1.4
	added type conversions to avoid warnings under codesys 3.0

hm	18. oct. 2008	rev 1.5
	using math constants

hm	17. dec. 2008	rev 1.6
	angles below horizon are displayed in negative degrees

hm	27. feb. 2009	rev 2.0
	new code with better accuracy

hm	7. mar. 2009	rev 2.1
	refraction is added after angle normalization
	deleted 10 second lockout
	added output for astronomical heigth h
*)

END_FUNCTION_BLOCK

// oscat_basic/POUs/Time&Date/REFRACTION
FUNCTION REFRACTION : REAL
VAR_INPUT
	ELEV : REAL;
END_VAR


(*
version 1.1	7. mar. 2009
programmer 	hugo
tested by		oscat

REFRACTION calculates the atmospheric refraction in degrees.
the input angle goes from 0 at the hirizon to 90 at midday.

*)

elev := LIMIT(-1.9, elev, 80.0);
REFRACTION := 0.0174532925199433 / TAN(0.0174532925199433 * (ELEV + 10.3 / (ELEV + 5.11)));


(* revision histroy
hm	14. jul. 2008	rev 1.0
	original release

hm	7. mar. 2009	rev 1.1
	using new formula

*)

END_FUNCTION

// oscat_basic/POUs/Time&Date/DAY_TO_TIME
FUNCTION DAY_TO_TIME : TIME
VAR_INPUT
	IN : REAL;
END_VAR


(*
version 1.1	24. feb. 2009
programmer 	hugo
tested by		tobias

converts an amount of days in real to time 
*)

DAY_TO_TIME := DWORD_TO_TIME(REAL_TO_DWORD(IN * 86400000.0));


(* revision history
hm	4. aug. 2006	rev 1.0
	original release

hm	24. feb. 2009	rev 1.1
	renamed input to IN
*)

END_FUNCTION

// oscat_basic/POUs/Time&Date/DAYS_DELTA
FUNCTION DAYS_DELTA : DINT
VAR_INPUT
	date_1 : DATE;
	date_2 : DATE;
END_VAR


(*
version 1.3		25. jan. 2011
programmer 		hugo
tested by		tobias

days_delta calculates the days between two dates. the days are calculated date_2 - date_1.

*)

IF DATE_1 > DATE_2 THEN
	DAYS_DELTA := - DWORD_TO_DINT((DATE_TO_DWORD(date_1) - DATE_TO_DWORD(date_2)) / 86400);
ELSE
	DAYS_DELTA := DWORD_TO_DINT((DATE_TO_DWORD(date_2) - DATE_TO_DWORD(date_1)) / 86400);
END_IF;

(* revision history
hm	27. dec 2006	rev 1.0
	original version

hm	16.9.2007		rev 1.1
	coorected an error in formula and changed algorithm to show positive and negative delta

hm	22. mar. 2008	rev 1.2
	changed output from int to dint because the total date range is 49710 days

hm	25. jan. 2011	rev 1.3
	improved performance
*)

END_FUNCTION

// oscat_basic/POUs/Time&Date/DAYS_IN_MONTH
FUNCTION DAYS_IN_MONTH : INT
VAR_INPUT
	IDATE : DATE;
END_VAR


(*
version 1.0	27. mar. 2009
programmer 	hugo
tested by		oscat

returs the total days of the current month. e.g. 31 for january.
the function works for dates from 1970 - 2099

*)

DAYS_IN_MONTH := DAY_OF_YEAR(IDATE);
IF LEAP_OF_DATE(IDATE) THEN
	CASE DAYS_IN_MONTH OF
		32..60	:	DAYS_IN_MONTH := 29;
		92..121 :	DAYS_IN_MONTH := 30;
		153..182:	DAYS_IN_MONTH := 30;
		245..274:	DAYS_IN_MONTH := 30;
		306..335:	DAYS_IN_MONTH := 30;
	ELSE
		DAYS_IN_MONTH := 31;
	END_CASE;
ELSE
	CASE DAYS_IN_MONTH OF
		32..59	:	DAYS_IN_MONTH := 28;
		91..120 :	DAYS_IN_MONTH := 30;
		152..181:	DAYS_IN_MONTH := 30;
		244..273:	DAYS_IN_MONTH := 30;
		305..334:	DAYS_IN_MONTH := 30;
	ELSE
		DAYS_IN_MONTH := 31;
	END_CASE;
END_IF;



(* revision history
hm	27. mar. 2009		rev 1.0
	original version

*)

END_FUNCTION

// oscat_basic/POUs/Time&Date/DAYS_IN_YEAR
FUNCTION DAYS_IN_YEAR : INT
VAR_INPUT
	IDATE : DATE;
END_VAR


(*
version 1.0	27. mar. 2009
programmer 	hugo
tested by		oscat

returs the total days of the year.
the function retruns 366 for leap years and 365 otherwise.
the function works for dates from 1970 - 2099


*)

IF LEAP_OF_DATE(IDATE) THEN
	DAYS_IN_YEAR := 366;
ELSE
	DAYS_IN_YEAR := 365;
END_IF;


(* revision history
hm	27. mar. 2009		rev 1.0
	original version

*)

END_FUNCTION

// oscat_basic/POUs/Time&Date/DCF77
FUNCTION_BLOCK DCF77
VAR_INPUT
	REC : BOOL;
	SET : BOOL;
	SDT : DT;
	DSI : BOOL;
END_VAR
VAR_INPUT CONSTANT
	SYNC_TIMEOUT : TIME := t#2m;
	TIME_OFFSET : INT := 1;
	DST_EN : BOOL := TRUE;
END_VAR
VAR_OUTPUT
	TP : BOOL;
	DS : BOOL;
	WDAY : INT;
	ERROR : BOOL := TRUE;
	RTC : DT;
	RTC1 : DT;
	MSEC : INT;
	SYNC : BOOL;
END_VAR
VAR
	mez : DT;
	utc : DT;
	state : INT;
	edge: BOOL;
	tx : TIME;
	ty: TIME;
	last : TIME;
	bits : ARRAY[0..58] OF BOOL;
	cnt : INT;
	i : INT;
	old_time : DT;
	minute : INT;
	hour : INT;
	day : INT;
	month : INT;
	year : INT;
	last_sync: TIME;
	t1: TIME;
	tz: TIME;
	init: BOOL;
END_VAR


(*
version 1.10	7. oct. 2008
programmer 	hugo
tested by	oscat

this is a decoder for a DCF77 signal.
the decoder decodes the DCF77 signal and checks for a valid Date_Time.
since the dcf77 signal is only secured with a simple parity the decoder waits for two consecutive valid transmissions before it sets the output signals.
given a valid reception by the receiver the decoder can take up to 3 minutes to start its clocks the first time.
after a valid signal is detected the error output goes low and dignals a valid dcf signal from the receiver.
a tp is only valid for one program cycle to allow for external rtc setting.
after a valid signal is detected two independent internal clocks are started (RTC and RTC1), the seconds  of these clocks are generated by software since the dcf signal is only valid for minutes.
rtc is always utc ( world time) and rtc1 can be set to any time zone by setting the time_zone_offset and enabling dst for automatic summertime.
a sync output signals the the rtc and rtc1 are in sync with the dcf77 signal, if the dcf77 signal is lost for more then the sync time the sync output goes low
but the rtc and rtc1 outputs keep running based on software timing until a valid dcf77 signal is received again and triggers the clock.
in addition a millisecond output gives further resolutionof the clocks.
a dst output shows if daylight saving time is enables and the weekday output shows which day of week currently is ( 1= monday ... 7= sunday).

*)

(* if tp was set it should only be active for 1 cycle *)
TP := FALSE;

(* read system time *)
t1 := DWORD_TO_TIME(T_PLC_MS());
tx := t1 - last;

IF rec XOR edge THEN
	edge := rec;
	IF NOT rec AND tx > t#1700ms AND tx < t#2000ms THEN
		(* start condition reached *)
		state := 0;
		tp := NOT error;
	ELSIF NOT rec AND tx > t#700ms AND tx < t#1000ms THEN
		(* second switch detected *)
		IF state < 58 THEN state := state +1; ELSE state := 0; END_IF;
	ELSIF rec AND tx  < t#120ms THEN
		(* bit 0 detected  *)
		bits[state] := 0;
	ELSIF rec AND tx > t#120ms AND tx < t#250ms THEN
		(* bit 1 detected *)
		bits[state] := 1;
	ELSE
		(* error condition received signal is not valid *)
		error := TRUE;
		state := 0;
	END_IF;
	last := last + tx;
	IF rec AND state = 58 THEN
		error := FALSE;

		(* decode the bits and check for possible errors *)
		IF bits[0] OR NOT (bits[17] XOR bits[18]) OR NOT bits[20] THEN error := TRUE; END_IF;
		(* decode minute *)
		MINUTE := 0;
		MINUTE.0 := bits[21];
		MINUTE.1 := bits[22];
		MINUTE.2 := bits[23];
		MINUTE.3 := bits[24];
		IF bits[25] THEN MINUTE := MINUTE + 10; END_IF;
		IF bits[26] THEN MINUTE := MINUTE + 20; END_IF;
		IF bits[27] THEN MINUTE := MINUTE + 40; END_IF;
		IF MINUTE > 59 OR (bits[21] XOR bits[22] XOR bits[23] XOR bits[24] XOR bits[25] XOR bits[26] XOR bits[27] XOR bits[28]) THEN error := TRUE; END_IF;

		(* decode hour *)
		HOUR := 0;
		HOUR.0 := bits[29];
		HOUR.1 := bits[30];
		HOUR.2 := bits[31];
		HOUR.3 := bits[32];
		IF bits[33] THEN HOUR := HOUR + 10; END_IF;
		IF bits[34] THEN HOUR := HOUR +20; END_IF;
		IF HOUR > 23 OR (bits[29] XOR bits[30] XOR bits[31] XOR bits[32] XOR bits[33] XOR bits[34] XOR bits[35]) THEN error := TRUE; END_IF;

		(* decode day of month *)
		day := 0;
		day.0 := bits[36];
		day.1 := bits[37];
		day.2 := bits[38];
		day.3 := bits[39];
		IF bits[40] THEN day := day + 10; END_IF;
		IF bits[41] THEN day := day + 20; END_IF;
		IF day > 31 THEN error := TRUE; END_IF;

		(* decode day of week *)
		wday := 0;
		wday.0 := bits[42];
		wday.1 := bits[43];
		wday.2 := bits[44];
		IF wday > 7 OR wday < 1 THEN error := TRUE; END_IF;

		(* decode month *)
		MONTH := 0;
		MONTH.0 := bits[45];
		MONTH.1 := bits[46];
		MONTH.2 := bits[47];
		MONTH.3 := bits[48];
		IF bits[49] THEN MONTH := MONTH +10; END_IF;
		IF MONTH > 12 THEN error := TRUE; END_IF;

		(* decode year *)
		YEAR := 0;
		YEAR.0 := bits[50];
		YEAR.1 := bits[51];
		YEAR.2 := bits[52];
		YEAR.3 := bits[53];
		IF bits[54] THEN YEAR := YEAR + 10; END_IF;
		IF bits[55] THEN YEAR := YEAR + 20; END_IF;
		IF bits[56] THEN YEAR := YEAR + 40; END_IF;
		IF bits[57] THEN YEAR := YEAR + 80; END_IF;

		(* check parity for bits 36 to 58 *)
		cnt := 0;
		FOR i := 36 TO 58 DO IF bits[i] THEN cnt := cnt + 1; END_IF; END_FOR;
		IF NOT EVEN(cnt) THEN error := TRUE; END_IF;

		(* time must be valid for two cycles to clear error flag *)
		IF NOT error THEN
			(* set outputs *)
			old_time := mez;
			IF YEAR >= 70 THEN YEAR := YEAR + 1900; ELSE YEAR := YEAR + 2000; END_IF;
			mez := SET_DT(YEAR,MONTH,day,HOUR,MINUTE,0);
			DS := bits[17];
			IF DS THEN
				UTC := DWORD_TO_DT(DT_TO_DWORD(mez) - 7200);
			ELSE
				UTC := DWORD_TO_DT(DT_TO_DWORD(mez) - 3600);
			END_IF;

			(* set trigger signal only if the receiver has received 2 successive minutes *)
			IF mez <> old_time + t#1m THEN error := TRUE ; END_IF;
		END_IF;
	END_IF;
END_IF;

(* this portion implements a free running clock which is triggered by the dcf77 signal *)
tz := DWORD_TO_TIME(INT_TO_DWORD(ABS(time_offset))* 3600000);

(* input sdt is copied to utc at first power up *)
IF NOT init OR SET THEN
	init := TRUE;
	utc := sdt;
	tp := TRUE;
	DS := DSI;
END_IF;

IF tp THEN
	rtc := utc;
	IF DS AND dst_en THEN
		IF time_offset < 0 THEN	rtc1 := rtc - tz + t#1h; ELSE rtc1 := rtc + tz + t#1h; END_IF;
	ELSE
		IF time_offset < 0 THEN rtc1 := rtc - tz; ELSE rtc1 := rtc + tz; END_IF;
	END_IF;
	sync := TRUE;
	last_sync := last;
	ty := last;
ELSIF rtc > DWORD_TO_DT(0) AND T1 - ty >= t#1s THEN
	rtc := rtc + t#1s;
	rtc1 := rtc1 + t#1s;
	ty := ty + t#1s;
	sync := ty - last_sync < sync_timeout AND last_sync > DWORD_TO_TIME(0);
	wday := DAY_OF_WEEK(DT_TO_DATE(rtc1));
	DS := dst_en AND DST(utc);
END_IF;
msec := TIME_TO_INT(t1 - ty);



(* decode information
bits		content
0			Bitwert immer 0
1 bis 14	reserviert für Betriebsinformationen (nicht für DCF77-Nutzer bestimmt)
15			Rufbit für Alarmierung der PTB-Mitarbeiter
			(bis Mai 2003: Bitwert = 0 falls normale Antenne in Verwendung; 1 = Backupantenne)
16			Bitwert = 1 falls ein Wechsel von MEZ nach MESZ oder umgekehrt bevorsteht; Dauer der Anzeige: 1 Stunde
17 + 18	gültige Zeit = MEZ, falls Bit 17=0 und Bit 18=1
			gültige Zeit = MESZ, falls Bit 17=1 und Bit 18=0
19			Bitwert = 1 falls innerhalb den nächsten 59 Minuten eine Schaltsekunde angeordnet ist. Beim Einfügen einer Schaltsekunde wird anstelle der 59. die 60. Sekundenmarke weggelassen und in der 58. erfolgt ausnahmsweise ein Trägerabfall.
20			Startbit für Zeitinformation (immer 1)
21 - 27		1, 2, 4, 8, 10, 20, 40 Minuten (bitweise Addition)
28			Prüfbit (gerade Parität) für die Bits 21-27
29 - 34		1, 2, 4, 8, 10, 20 Stunden (bitweise Addition)
35			Prüfbit (gerade Parität) für die Bits 29-34
36 - 41		Tagesnummer im aktuellen Monat: 1, 2, 4, 8, 10, 20 (bitweise Addition)
42 - 44		Tagesnummer in der aktuellen Woche: 1, 2, 4 (bitweise Addition)
45 - 49		Monatsnummer: 1, 2, 4, 8, 10 (bitweise Addition)
50 - 57		Jahr (zweistellig): 1, 2, 4, 8, 10, 20, 40, 80 (bitweise Addition)
58			Prüfbit (gerade Parität) füR die Bits 36-57

*)
(* revision history

hm 2.feb 2007		rev 1.1
	change wday and dst outputs when there is no dcf reception

hm	26.feb 2007		rev 1.2
	changed statements where t#1h would be substracted from DT.
	under certain conditions the compiler would crash translating this statement

hm	17. sep 2007	rev 1.3
	replaced time() with T_PLC_MS() for compatibility reasons

hm	24. oct 2007		rev 1.4
	changed dst calculation because function dst was upgraded no error in DCF77 only a change in DST

hm	12. nov 2007		rev 1.5
	changed time_offset from time to integer to allow for negative offset time zones

hm	8. dec 2007		rev 1.6
	corrected an error in time_zone calculation

hm 23. jan 2008		rev 1.7
	added sdt input which is used to initialize rtc and rtc1 during first cycle.

hm 16. mar 2008		rev 1.8
	changed output weekday to wday and dst to ds for compatibility reasons

hm	19. apr. 2008	rev 1.9
	added input dsi to allow to set daylight savings time when SDT is TRUE.
	added asynchronous SET input

hm	7. oct. 2008	rev 1.10
	changed function weekday to day_of_week

*)

END_FUNCTION_BLOCK

// oscat_basic/POUs/Time&Date/DT_TO_SDT
FUNCTION DT_TO_SDT : SDT
VAR_INPUT
	DTI : DT;
END_VAR
VAR
	tmp : DATE;
	tdt : DWORD;
END_VAR


(*
version 1.0	18. oct 2008
programmer 	hugo
tested by	oscat

converts date_time to Structured date time (SDT)

*)

tmp := DT_TO_DATE(dti);
tdt := DT_TO_DWORD(dti) - DATE_TO_DWORD(tmp);
DT_TO_SDT.YEAR := YEAR_OF_DATE(tmp);
DT_TO_SDT.MONTH := MONTH_OF_DATE(tmp);
DT_TO_SDT.DAY := DAY_OF_MONTH(tmp);
DT_TO_SDT.WEEKDAY := DAY_OF_WEEK(tmp);
DT_TO_SDT.SECOND := DWORD_TO_INT(tdt MOD 60);
DT_TO_SDT.MINUTE := DWORD_TO_INT((tdt / 60) MOD 60);
DT_TO_SDT.HOUR := DWORD_TO_INT(tdt / 3600);

(* revision history

hm 18. oct. 2008	rev 1.0
	original version

*)

END_FUNCTION

// oscat_basic/POUs/Time&Date/DT2_TO_SDT
FUNCTION DT2_TO_SDT : SDT
VAR_INPUT
	DI : DATE;
	TI : TOD;
END_VAR


(*
version 1.0	18. oct 2008
programmer 	hugo
tested by	oscat

converts date and time of day to Structured date time (SDT)

*)

DT2_TO_SDT.YEAR := YEAR_OF_DATE(di);
DT2_TO_SDT.MONTH := MONTH_OF_DATE(di);
DT2_TO_SDT.DAY := DAY_OF_MONTH(di);
DT2_TO_SDT.WEEKDAY := DAY_OF_WEEK(di);
DT2_TO_SDT.MS := DWORD_TO_INT(TOD_TO_DWORD(ti) MOD 1000);
DT2_TO_SDT.SECOND := DWORD_TO_INT((TOD_TO_DWORD(ti) / 1000) MOD 60);
DT2_TO_SDT.MINUTE := DWORD_TO_INT((TOD_TO_DWORD(ti) / 60000) MOD 60);
DT2_TO_SDT.HOUR := DWORD_TO_INT(TOD_TO_DWORD(ti) / 3600000);

(* revision history

hm 18. oct. 2008	rev 1.0
	original version

*)

END_FUNCTION

// oscat_basic/POUs/Time&Date/HOUR_OF_DT
FUNCTION HOUR_OF_DT : INT
VAR_INPUT
	XDT : DT;
END_VAR


(*
	version 1.0	6. jun. 2008
	programmer 	oscat
	tested BY	oscat

HOUR_OF_DT returns the current hour (hour of the day) of a DT variable

*)

HOUR_OF_DT := DWORD_TO_INT((DT_TO_DWORD(XDT) MOD 86400) / 3600);


(* revision history
hm		6.9.2008	rev 1.0
	original version


*)

END_FUNCTION

// oscat_basic/POUs/Time&Date/JD2000
FUNCTION JD2000 : REAL
VAR_INPUT
	DTI : DT;
END_VAR


(*
version 1.0	15. jul. 2008
programmer 	hugo
tested by	oscat

JULIAN calculates the astronomic julian date from 1.1.2000-12:00.

*)

JD2000 := DWORD_TO_REAL(DT_TO_DWORD(DTI) - 946728000) / 86400.0;

(* revision histroy
hm	15. jul. 2008	rev 1.0
	original release


*)

END_FUNCTION

// oscat_basic/POUs/Time&Date/LEAP_DAY
FUNCTION LEAP_DAY : BOOL
VAR_INPUT
	IDATE : DATE;
END_VAR
VAR
END_VAR


(*
version 1.2	24. jan. 2011
programmer 	hugo
tested by	oscat


leap_day is true if the tested day is a leap day (29. of february).  
  
*)

LEAP_DAY := DATE_TO_UDINT(IDATE) MOD 126230400 = 68169600;


(* change history

hm 	15. jun. 2008	rev 1.0
	original version

hm	7. oct. 2008	rev 1.1
	changed function month to month_of_date

hm	24. jan. 2011	rev 1.2
	improved performance
*)

END_FUNCTION

// oscat_basic/POUs/Time&Date/LTIME_TO_UTC
FUNCTION LTIME_TO_UTC : DT
VAR_INPUT
	CONVERSION_LTIME : DT;
	DST : BOOL;
	TIME_ZONE_OFFSET : INT;
END_VAR


(*
version 1.7	13. nov. 2009
programmer 	hugo
tested by		oscat

LTIME_TO_UTC calculates UTC (World Time) from a local time LTIME. utc is calculated 
by subtracting Time_Zone_Offset from ltime and if dst it true subtracting an additional hour from ltime.

*)

LTIME_TO_UTC := UDINT_TO_DT(DT_TO_UDINT(CONVERSION_LTIME) - INT_TO_UDINT(TIME_ZONE_OFFSET) * 60);
IF DST THEN LTIME_TO_UTC := LTIME_TO_UTC - T#1h; END_IF;

(* revision history
hm 5.7.2007		rev 1.0		
	original version

hm 5.11.2007		rev 1.1
	replaced literal constant with variable because of error in möller ecp4 compiler

hm	12.nov 2007	rev 1.2
	changed Type of time_zone_offset from time to int to allow for time zones with negative offset

hm	8. dec 2007	rev 1.3
	corrected a problem with time_zone_offset

hm	14. oct. 2008	rev 1.4
	changed time_zone_offset from int to real to allow for half hour offset

hm	20. oct. 2006	rev 1.5
	changed time_zone_offset from Real to INT, now in Minutes

hm	27. feb. 2009	rev 1.6
	added type conversions to avoid warnings under codesys 3.0

ks	13. nov. 2009	rev 1.7
	corrected error in formula

*)

END_FUNCTION

// oscat_basic/POUs/Time&Date/MINUTE_OF_DT
FUNCTION MINUTE_OF_DT : INT
VAR_INPUT
	XDT : DT;
END_VAR


(*
	version 1.0	6. jun. 2008
	programmer 	oscat
	tested BY	oscat

MINUTE_OF_DT returns the current minute (minute of the hour) of a DT variable

*)

MINUTE_OF_DT := DWORD_TO_INT(DT_TO_DWORD(XDT) MOD 3600) / 60;


(* revision history
hm		6.9.2008	rev 1.0
	original version


*)

END_FUNCTION

// oscat_basic/POUs/Time&Date/MINUTE_TO_TIME
FUNCTION MINUTE_TO_TIME : TIME
VAR_INPUT
	IN : REAL;
END_VAR


(*
version 1.2	24. feb. 2009
programmer 	hugo
tested by		oscat

converts an amount of minutes in real to time

*)

MINUTE_TO_TIME := DWORD_TO_TIME(REAL_TO_DWORD(IN * 60000.0));


(* revision history
hm	4. aug 2006	rev 1.0
	original version

hm	14. mar 2008	rev 1.1
	rounded the input after the last digit

hm	24. feb. 2009	rev 1.2
	changed input to IN

*)

END_FUNCTION

// oscat_basic/POUs/Time&Date/MONTH_BEGIN
FUNCTION MONTH_BEGIN : DATE
VAR_INPUT
	idate : DATE;
END_VAR


(*
version 1.0	15. jun. 2008
programmer 	hugo
tested by	oscat

returns the date for the first day of the current month in the current year.

*)

MONTH_BEGIN := DWORD_TO_DATE(DATE_TO_DWORD(idate) - INT_TO_DWORD(DAY_OF_MONTH(idate) - 1) * 86400);

(* revision history
hm	15. jun. 2008	rev 1.0
	original version	

*)

END_FUNCTION

// oscat_basic/POUs/Time&Date/MONTH_END
FUNCTION MONTH_END : DATE
VAR_INPUT
	IDATE : DATE;
END_VAR


(*
version 1.1	7. oct. 2008
programmer 	hugo
tested by	oscat

returns the date for the last day of the current month in the current year.

*)

MONTH_END := DWORD_TO_DATE(DATE_TO_DWORD(SET_DATE(YEAR_OF_DATE(idate),MONTH_OF_DATE(idate)+1,1)) - 86400);



(* revision history
hm	15. jun. 2008	rev 1.0
	original version	

hm	7. oct. 2008	rev 1.1
	changed function year to year_of_date
	changed function month to month_of_date

*)

END_FUNCTION

// oscat_basic/POUs/Time&Date/PERIOD2
FUNCTION PERIOD2 : BOOL
VAR_INPUT
	DP : ARRAY[0..3,0..1] OF DATE;
	DX : DATE;
END_VAR


(*
version 1.0	27. apr. 2008
programmer 	hugo
tested by	tobias

PERIOD2 checks if DX is within one of 4 periods and sets the output true if so.

*)

PERIOD2 := 	(DX >= DP[0,0] AND DX <= DP[0,1]) OR
			(DX >= DP[1,0] AND DX <= DP[1,1]) OR
			(DX >= DP[2,0] AND DX <= DP[2,1]) OR
			(DX >= DP[3,0] AND DX <= DP[3,1]);


(* revision history

hm		27. apr 2008	rev 1.0
	original version


*)

END_FUNCTION

// oscat_basic/POUs/Time&Date/RTC_2
FUNCTION_BLOCK RTC_2
VAR_INPUT
	SET : BOOL;
	SDT : DT;
	SMS : INT;
	DEN : BOOL;
	OFS : INT;
END_VAR
VAR_OUTPUT
	UDT : DT;
	LDT : DT;
	DSO : BOOL;
	XMS : INT;
END_VAR
VAR
	RT : RTC_MS;
END_VAR

(*
version 1.4	27. 	apr. 2011
programmer 	hugo
tested by		tobias

RTC_2 is a real time clock module which runs utc and generates local time from utc.
daylight savings time can be enabled with den and an additional local time is generated with a delay of ofs im minutes.

*)

(* call rtc *)
RT(SET := SET, SDT := SDT, SMS := SMS);
UDT := rt.xdt;
XMS := rt.XMS;

(* check for daylight savings time and set dso output *)
DSO := DST(udt) AND DEN;

(* calculate time offset and set ldt output *)
LDT := DWORD_TO_DT(DT_TO_DWORD(UDT) + INT_TO_DWORD(ofs + BOOL_TO_INT(DSO)*60) * 60);


(* revision history
hm		20. jan. 2008	rev 1.0
	original version

hm		20. feb. 2008	rev 1.1
	added Millisecond Set input

hm		12. jun. 2008	rev 1.2
	improved performance

hm		20. jan. 2011	rev 1.3
	changed offset to be in minutes

hm		27. apr. 2011	rev 1.4
	fixed error with local time calculation

*)

END_FUNCTION_BLOCK

// oscat_basic/POUs/Time&Date/RTC_MS
FUNCTION_BLOCK RTC_MS
VAR_INPUT
	SET : BOOL;
	SDT : DT;
	SMS : INT;
END_VAR
VAR_OUTPUT
	XDT : DT;
	XMS : INT;
END_VAR
VAR
	init: BOOL;
	last: DWORD;
	Tx: DWORD;
END_VAR

(*
version 1.1	20. feb. 2008
programmer 	hugo
tested by	tobias

RTC_MS is a real time clock module which can be set to SDT when set is TRUE and the outputs XDT and XT present the DateTime and TOD with a resolution of milliseconds.

*)

tx := T_PLC_MS();
IF set OR NOT init THEN
	(* clock needs to be set when set is true or after power up *)
	init := TRUE;
	xdt := SDT;
	XMS := SMS;
ELSE
	XMS := XMS + DWORD_TO_INT(tx - last);
	(* check if one second has expired *)
	IF XMS > 999 THEN
		XDT := XDT + T#1s;
		XMS := XMS - 1000;
	END_IF;
END_IF;
last := tx;


(* revision history
hm		20. jan. 2008	rev 1.0
	original version

hm		20. feb. 2008	rev 1.1
	added Millisecond Set input
*)

END_FUNCTION_BLOCK

// oscat_basic/POUs/Time&Date/SDT_TO_DATE
FUNCTION SDT_TO_DATE : DATE
VAR_INPUT
	DTI : SDT;
END_VAR


(*
version 1.0	18. oct 2008
programmer 	hugo
tested by	oscat

converts Structured date time (SDT) to Date Time

*)

SDT_TO_DATE := SET_DATE(DTI.YEAR, DTI.MONTH, DTI.DAY);



(* revision history

hm 18. oct. 2008	rev 1.0
	original version

*)

END_FUNCTION

// oscat_basic/POUs/Time&Date/SDT_TO_DT
FUNCTION SDT_TO_DT : DT
VAR_INPUT
	DTI : SDT;
END_VAR


(*
version 1.0	18. oct 2008
programmer 	hugo
tested by	oscat

converts Structured date time (SDT) to Date Time

*)

SDT_TO_DT := SET_DT(DTI.YEAR, DTI.MONTH, DTI.DAY, DTI.HOUR, DTI.MINUTE, DTI.SECOND);



(* revision history

hm 18. oct. 2008	rev 1.0
	original version

*)

END_FUNCTION

// oscat_basic/POUs/Time&Date/SDT_TO_TOD
FUNCTION SDT_TO_TOD : TOD
VAR_INPUT
	DTI : SDT;
END_VAR


(*
version 1.1	16. nov. 2008
programmer 	hugo
tested by	oscat

converts Structured date time (SDT) to Date Time

*)

SDT_TO_TOD := DWORD_TO_TOD(INT_TO_DWORD(DTI.HOUR) * 3600000 + INT_TO_DWORD(DTI.MINUTE) * 60000 + INT_TO_DWORD(DTI.SECOND) * 1000 + INT_TO_DWORD(DTI.MS));



(* revision history

hm 18. oct. 2008	rev 1.0
	original version

hm	16. nov. 2008	rev 1.1
	added typecasts to avoid warnings
*)

END_FUNCTION

// oscat_basic/POUs/Time&Date/SECOND_OF_DT
FUNCTION SECOND_OF_DT : INT
VAR_INPUT
	XDT : DT;
END_VAR


(*
	version 1.0	6. jun. 2008
	programmer 	oscat
	tested BY	oscat

SECOND_OF_DT returns the current second (second of minute) of a DT variable

*)

SECOND_OF_DT := DWORD_TO_INT(DT_TO_DWORD(XDT) MOD 60);

(* revision history
hm		6.9.2008	rev 1.0
	original version

*)

END_FUNCTION

// oscat_basic/POUs/Time&Date/SECOND_TO_TIME
FUNCTION SECOND_TO_TIME : TIME
VAR_INPUT
	IN : REAL;
END_VAR


(*
version 1.2	24. feb. 2009
programmer 	hugo
tested by		tobias

converts an amount of seconds in real to time
execution TIME on wago 750-841 =  17us 

*)

SECOND_TO_TIME := DWORD_TO_TIME(REAL_TO_DWORD(IN * 1000.0));

(* revision history
hm	4. aug. 2006	rev 1.0
	original version

hm	14. mar. 2008	rev 1.1
	rounded the input after the last digit

hm	24. feb. 2009	rev 1.2
	changed input to IN
*)

END_FUNCTION

// oscat_basic/POUs/Time&Date/SET_TOD
FUNCTION SET_TOD : TOD
VAR_INPUT
	hour : INT;
	minute : INT;
	second : REAL;
END_VAR


(*
version 1.5	16. mar 2008
programmer 	hugo
tested by	tobias

creates tod from hour minute and second 

*)

SET_TOD := DWORD_TO_TOD(REAL_TO_DWORD(SECOND * 1000.0) + INT_TO_DWORD(MINUTE) * 60000 + INT_TO_DWORD(HOUR) * 3600000);

(* revision history

hm		4.aug.2006		rev 1.0
	original version

hm		11. sep 2007	rev 1.1
	changed coding to avoid a compiler warning under twincat.

hm		1. nov 2007	rev 1.2
	changed coding to avoid possible overrun situation on möller ecp4

hm		2. Nov	2007	rev 1.3
	changed dword to DINT in calcualtion to avoid warnings with some compilers

hm		14. mar 2008	rev 1.4
	changed code to avoid rounding problem at last digit of millisecond

hm		16. mar. 2008	rev 1.5
	added type conversions to avoid warning under codesys 3.0
*)

END_FUNCTION

// oscat_basic/POUs/Time&Date/TIMECHECK
FUNCTION TIMECHECK : BOOL
VAR_INPUT
	TD : TOD;
	START : TOD;
	STOP : TOD;
END_VAR


(*
version 1.0	19. jul. 2009
programmer 	oscat
tested by		oscat

this function retruns true if the daytime TD is between start and stop and returns true if so.
if you want to generate an event to span over midnight, start timemust be later than the stop time.

*)

IF stop < start THEN
	TIMECHECK := start <= TD OR TD < stop;
ELSE
	TIMECHECK := start <= TD AND TD < stop;
END_IF;



(* revision history
hm 19. jul. 2009	rev 1.0
	original release

*)

END_FUNCTION

// oscat_basic/POUs/Time&Date/TON_P
FUNCTION_BLOCK TON_P	// Ton pausable
(* If IN is FALSE, Q is FALSE and ET is 0. As soon as IN becomes TRUE, 
the time will begin to be counted in milliseconds in ET until its value is equal to PT. 
It will then remain constant. Q is TRUE when IN is TRUE and ET is equal to PT. 
Otherwise it is FALSE. Thus, Q has a rising edge when the time indicated in PT in milliseconds has run out. 
PAUSE allows for pausing the timer while retaining the elapsed time. 
The timer will thus continue with the same amount of time left before pausing. *)
VAR_INPUT
    IN : BOOL;		(* starts timer with rising edge, resets timer with falling edge *)
    PT : TIME;		(* time to pass, before Q is set *)
    PAUSE : BOOL;
END_VAR
VAR_OUTPUT
    Q : BOOL;		(* is TRUE, PT seconds after IN had a rising edge *)
    ET : TIME;		(* elapsed time *)
END_VAR
VAR
    rtPause : R_TRIG;	(* rising edge trigger *)
    tTimePaused : TIME;
    ton : TON;		(* timer on-delay *)
END_VAR

IF NOT IN THEN
    tTimePaused := T#0S;
END_IF

rtPause(CLK := IN AND PAUSE);

IF rtPause.Q THEN
    tTimePaused := tTimePaused + ton.ET;
END_IF

ton(IN := IN AND NOT PAUSE, PT := PT - tTimePaused);

//IF ET >= PT THEN
//	Q := TRUE;
//ELSE
//	Q := FALSE;
//END_IF

Q := ton.Q;

ET := tTimePaused + ton.ET;

END_FUNCTION_BLOCK

// oscat_basic/POUs/Time&Date/YEAR_END
FUNCTION YEAR_END : DATE
VAR_INPUT
	y : INT;
END_VAR


(*
version 1.1	24. jan. 2011
programmer 	hugo
tested by	oscat

returs the date of december 31st for the given year  
the function works for dates from 1970 - 2099 

*)

YEAR_END := DWORD_TO_DATE(SHR(INT_TO_DWORD(y) * 1461 - 2876712, 2) * 86400);



(* revision history
hm	15. jun. 2008	rev 1.0
	original version

hm	24. jan 2011	rev 1.1
	improved performance
*)

END_FUNCTION

// oscat_building/POUs/actuators/ACTUATOR_2P
FUNCTION_BLOCK ACTUATOR_2P
VAR_INPUT
	IN : BYTE;
	TEST : BOOL;
	ARE : BOOL := TRUE;
END_VAR
VAR_IN_OUT
	ARX : BOOL;
END_VAR
VAR_INPUT CONSTANT
	CYCLE_TIME : TIME;
	SENS : BYTE;
	SELF_ACT_TIME : TIME;
	SELF_ACT_PULSE : TIME;
	SELF_ACT_CYCLES : INT := 1;
END_VAR
VAR_OUTPUT
	OUT : BOOL;
	ARO : BOOL;
END_VAR
VAR
	timer : AUTORUN;
	pwgen : GEN_PULSE;
END_VAR


(*
version 2.1	24. jan. 2009
programmer 	hugo
tested by		oscat

this is an intelligent actuator interface for any 2point actuator like coil drive.
the 2Point actuator can only switch on/off and therefore the input must be converted to on/off cycles.
the interface can be programmed with double click on the symbol.
in addition a self_act_time and self_act_cycles ca be programmed to switch n times on/off every self_act_time to avoid a valve to freeze.
the input value must be between 0 and 255. with the setup variable sens one can specify what must be the minimum input to turn the valve on at all.
at the same time an input > 255-sens will turn the valve on at all times.


*)

(* run the autorun timer *)
timer(trun := SELF_ACT_PULSE * (2 * SELF_ACT_CYCLES), toff := SELF_ACT_TIME, Test := TEST, ARE := ARE, arx := ARX);
ARO := timer.ARO;

(* run the pulse width generator *)
IF aro THEN
	pwgen(PTL := SELF_ACT_PULSE, PTH := SELF_ACT_PULSE);
	out := pwgen.Q;
ELSIF in < sens THEN
	out := FALSE;
ELSIF in > BYTE#255 - sens THEN
	out := TRUE;
ELSE
	pwgen.PTH := (CYCLE_TIME * BAND_B(IN,SENS)) / 255;
	pwgen.PTL := CYCLE_TIME - pwgen.PTH;
	pwgen();
	out := pwgen.Q;
END_IF;



(* revision history
hm	7.10.2006 		rev 1.1
	changed error pos could not reach 1 or 0 under certain conditions due to error in code.
	changed on and off in force and force_in for better usability.

hm	17.1.2007		rev 1.2
	deleted unused variable time_overflow

hm	15.9.2007		rev 1.3
	replaced time() with T_PLC_MS for compatibility and performance reasons

hm	19. 11 2007		rev 1.4
	replaced left over statement time() with tx

hm	27. 12. 2007	REV 1.5
	CHANGED CODE FOR BETTER PERFORMANCE

hm	21. oct. 2008	rev 1.6
	code optimized

hm	23. nov. 2008	rev 2.0
	new code using library modules

hm	24. jan. 2009	rev 2.1
	deleted unused var inb
*)

END_FUNCTION_BLOCK

// oscat_building/POUs/actuators/AUTORUN
FUNCTION_BLOCK AUTORUN
VAR_INPUT
	IN : BOOL;
	TEST : BOOL;
	ARE : BOOL := TRUE;
END_VAR
VAR_IN_OUT
	ARX : BOOL;
END_VAR
VAR_INPUT CONSTANT
	TRUN : TIME;
	TOFF : TIME;
END_VAR
VAR_OUTPUT
	OUT : BOOL;
	ARO : BOOL;
END_VAR
VAR
	timer : _RMP_B;
	val : BYTE;
END_VAR



(*
version 1.0	20. nov 2008
programmer 	hugo
tested by	oscat




*)

(* run the integrator when T_off > T#0s *)
IF TOFF > T#0s THEN
	timer(DIR:= OUT, TR := SEL(OUT, TOFF, TRUN), RMP := val);
ELSE
	val := 255;
END_IF;


(* when timer = 0 or test then initiate autorun until timer reaches 255 *)
IF (NOT ARX AND ARE AND val = 0) OR TEST THEN
	val := 0;
	ARO := TRUE;
	ARX := TRUE;
ELSIF val = 255 AND ARO THEN
	ARO := FALSE;
	ARX := FALSE;
END_IF;

(* output is true when autorun ARO is true or in = TRUE *)
out := IN OR ARO;



(* revision history
hm 20. nov. 2008	rev 1.0
	original version

*)

END_FUNCTION_BLOCK

// oscat_building/POUs/electrical/CLICK
FUNCTION_BLOCK CLICK
VAR_INPUT
	in : BOOL;
END_VAR
VAR_OUTPUT
	Q : BOOL;
	single : BOOL;
	double : BOOL;
	triple : BOOL;
	status: BYTE;
END_VAR
VAR_INPUT CONSTANT
	T_debounce : TIME := t#10ms;
	T_short : TIME := t#200ms;
	T_pause : TIME := t#500ms;
	T_reconfig : TIME := t#1m;
END_VAR
VAR
	s_in : SW_RECONFIG;
	tx: TIME;
	state: INT;
	last: TIME;
END_VAR

(*
version 2.0	28. dec. 2008
programmer 	oscat
tested by		oscat

click checks an input for single, double or tripple click and sets the corresponding output single, doulbe or triple for the time the input stays high at the last click.
the maximum high and low time for a click can be configured with setup variables.
the input configures itself to be high or low active depending on which state the input stays longer than t_reconfig.

*)

(* reconfiguration and debounce circuitry *)
s_in(in := in, TD := T_debounce, TR := T_reconfig);

(* read system time *)
tx := DWORD_TO_TIME(T_PLC_MS());

(* count the mumber of clicks *)
IF s_in.Q XOR Q THEN
	last := tx;
	IF s_in.Q THEN state := state + 1; END_IF;
END_IF;
Q := s_in.Q;

(* set outputs *)
IF state > 0 THEN
	IF (Q AND tx - last > t_short) OR (NOT Q AND tx - last > t_pause) THEN
		CASE state OF
			1:	single := TRUE;
				status := 111;
			2:	double := TRUE;
				status := 112;
			3:	triple := TRUE;
				status := 113;
		END_CASE;
		state := 0;
	END_IF;
ELSIF NOT q THEN
	single := FALSE;
	double := FALSE;
	triple := FALSE;
	status := 110;
	last := tx;
	state := 0;
END_IF;





(* revision history

15 Feb 2007	rev 1.0	hm
	created original version

18.5.2007	rev 1.1 hm
	corrected an error while execution would stop after t_reconfig elapsed.

15.9.2007	rev 1.2 hm
	replaced Time() with T_PLC_MS for compatibility and performance reasons

28. dec. 2008	rev 2.0
	rewritten using modular approach

*)

END_FUNCTION_BLOCK

// oscat_building/POUs/electrical/DEBOUNCE
FUNCTION_BLOCK DEBOUNCE
VAR_INPUT
	IN : BOOL;
	TD : TIME;
	PM : BOOL;
END_VAR

VAR_OUTPUT
	Q : BOOL;
END_VAR
VAR
	deb : TOF;
END_VAR

(*
version 1.0	22. sep. 2008
programmer 	oscat
tested by	tobias

DEBOUNCE is used to debounce switch inputs.
in addition to the debounce functionality this FB can also be used to detect rising edges on IN when PM = TRUE.
When PM = FALSE, Q follows in with the debounce functionality.

*)


